KUKA KRL program: EPS_2_251315_MH01A_A_20251126070854.src

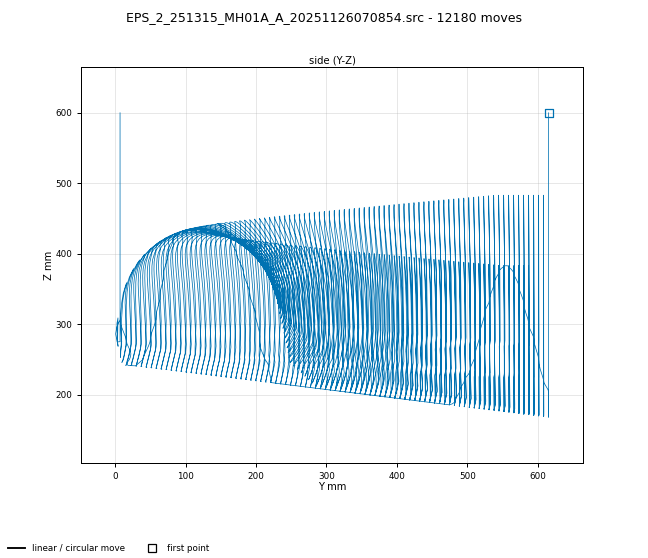
[picture p0: tool path of EPS_2_251315_MH01A_A_20251126070854.src, 12180 of 12182 moves have a stored position in this frame; points joined in program order, loops and branches not executed]
&ACCESS RVP
&REL 4
&COMMENT QRS 19112012
&PARAM EDITMASK = *
DEF PART()
EXT BAS (BAS_COMMAND :IN,REAL :IN )
INT I
BAS (#INITMOV,0 )

;KUKA QRS Post kuka4.cps  Date:22-06-2017 !

File_ID=2929

QRS_PRE_INIT()

;Init var - Until changes are made in qrs_pre_init
Outlet_Square_prg=0
Inlet_1_Square_prg=0
Inlet_2_Square_prg=0
Inlet_3_Square_prg=0
Inlet_4_Square_prg=0
Inlet_5_Square_prg=0

Outlet_1={X 0.000, Y 540.910, Z 382.500, B 0.000, E1 0.000 }
Inlet_1={X 0.000, Y 548.330, Z 308.000, B 0.000, E1 110.000 }
Outlet_1_type=201
Inlet_1_type=150
;QRS#1=Sidecore dimensions
;QRS#2=200-8" PVC SDR 35
;QRS#3=150-6" PVC SDR 28
;QRS#4=
;QRS#5=
;QRS#6=
;QRS#7=
;QRS#8=
;QRS#9=12-08 PSX
;QRS#10=10-06 PSX
;QRS#11=
;QRS#12=
;QRS#13=
;QRS#14=
;QRS#15=
;QRS#16=1220x127x762 2,5'
;QRS#17=EPS Height
;QRS#18=483
;QRS#19=*
;QRS#20= UPDATED VERSION 22-06-2017
;QRS#21=*
Outlet_Square=0100
Inlet_1_Square=070
Inlet_2_Square=0
Inlet_3_Square=0
Inlet_4_Square=0
Inlet_5_Square=0
Mill_Square=1
Outlet_Square_Prg=204
Inlet_1_Square_prg=203

QRS_INIT()

$ADVANCE=5

; T1
PTP {E1 173.696,E2 173.696}
PTP {X 0,Y 615.498,A -85,B 0,C 180,E1 173.696,E2 173.696,E3 0,E4 0,E5 0,E6 0}
QRS_SPEED_INIT()
LIN {X 0,Y 615.498,Z 600,A -85,B 0,C 180,E1 173.696,E2 173.696,E3 0,E4 0,E5 0,E6 0} C_VEL
LIN {X 0,Y 615.498,Z 213.72,A -85,B 0,C 180,E1 173.696,E2 173.696} C_VEL
LIN {X 0,Y 615.498,Z 205.494,A -85,B 0,C 180,E1 173.696,E2 173.696} C_VEL
LIN {X 0,Y 615.487,Z 203.734,A -85,B 0,C 180,E1 173.422,E2 173.422} C_VEL
LIN {X 0,Y 615.486,Z 220.973,A -85,B 0,C 180,E1 170.47,E2 170.47} C_VEL
LIN {X 0,Y 615.484,Z 223.487,A -85,B 0,C 180,E1 170.097,E2 170.097} C_VEL
LIN {X 0,Y 615.48,Z 225.832,A -85,B 0,C 180,E1 170.034,E2 170.034} C_VEL
LIN {X 0,Y 615.49,Z 299.844,A -85,B 0,C 180,E1 169.155,E2 169.155} C_VEL
LIN {X 0,Y 615.497,Z 309.209,A -85,B 0,C 180,E1 168.959,E2 168.959} C_VEL
LIN {X 0,Y 615.498,Z 318.215,A -85,B 0,C 180,E1 168.682,E2 168.682} C_VEL
LIN {X 0,Y 615.499,Z 327.343,A -85,B 0,C 180,E1 168.307,E2 168.307} C_VEL
LIN {X 0,Y 615.495,Z 338.158,A -85,B 0,C 180,E1 167.722,E2 167.722} C_VEL
LIN {X 0,Y 615.496,Z 346.444,A -85,B 0,C 180,E1 167.135,E2 167.135} C_VEL
LIN {X 0,Y 615.5,Z 354.141,A -85,B 0,C 180,E1 166.463,E2 166.463} C_VEL
LIN {X 0,Y 615.497,Z 360.745,A -85,B 0,C 180,E1 165.758,E2 165.758} C_VEL
LIN {X 0,Y 615.495,Z 366.931,A -85,B 0,C 180,E1 164.944,E2 164.944} C_VEL
LIN {X 0,Y 615.492,Z 372.054,A -85,B 0,C 180,E1 164.095,E2 164.095} C_VEL
LIN {X 0,Y 615.498,Z 376.623,A -85,B 0,C 180,E1 163.072,E2 163.072} C_VEL
LIN {X 0,Y 615.487,Z 379.784,A -85,B 0,C 180,E1 162.043,E2 162.043} C_VEL
LIN {X 0,Y 615.487,Z 381.203,A -85,B 0,C 180,E1 161.354,E2 161.354} C_VEL
LIN {X 0,Y 615.491,Z 382.08,A -85,B 0,C 180,E1 160.663,E2 160.663} C_VEL
LIN {X 0,Y 615.492,Z 382.389,A -85,B 0,C 180,E1 159.968,E2 159.968} C_VEL
LIN {X 0,Y 615.496,Z 382.089,A -85,B 0,C 180,E1 159.27,E2 159.27} C_VEL
LIN {X 0,Y 615.493,Z 381.22,A -85,B 0,C 180,E1 158.569,E2 158.569} C_VEL
LIN {X 0,Y 615.492,Z 379.266,A -85,B 0,C 180,E1 157.653,E2 157.653} C_VEL
LIN {X 0,Y 615.492,Z 376.497,A -85,B 0,C 180,E1 156.801,E2 156.801} C_VEL
LIN {X 0,Y 615.492,Z 371.558,A -85,B 0,C 180,E1 155.729,E2 155.729} C_VEL
LIN {X 0,Y 615.494,Z 366.205,A -85,B 0,C 180,E1 154.864,E2 154.864} C_VEL
LIN {X 0,Y 615.493,Z 360.324,A -85,B 0,C 180,E1 154.103,E2 154.103} C_VEL
LIN {X 0,Y 615.495,Z 353.723,A -85,B 0,C 180,E1 153.406,E2 153.406} C_VEL
LIN {X 0,Y 615.485,Z 344.747,A -85,B 0,C 180,E1 152.639,E2 152.639} C_VEL
LIN {X 0,Y 615.495,Z 335.257,A -85,B 0,C 180,E1 152.019,E2 152.019} C_VEL
LIN {X 0,Y 615.499,Z 326.105,A -85,B 0,C 180,E1 151.548,E2 151.548} C_VEL
LIN {X 0,Y 615.498,Z 317.502,A -85,B 0,C 180,E1 151.203,E2 151.203} C_VEL
LIN {X 0,Y 615.498,Z 308.063,A -85,B 0,C 180,E1 150.923,E2 150.923} C_VEL
LIN {X 0,Y 615.484,Z 298.594,A -85,B 0,C 180,E1 150.735,E2 150.735} C_VEL
LIN {X 0,Y 615.478,Z 223.968,A -85,B 0,C 180,E1 149.84,E2 149.84} C_VEL
LIN {X 0,Y 615.481,Z 222.831,A -85,B 0,C 180,E1 149.745,E2 149.745} C_VEL
LIN {X 0,Y 615.475,Z 206.472,A -85,B 0,C 180,E1 146.959,E2 146.959} C_VEL
LIN {X 0,Y 615.468,Z 191.559,A -85,B 0,C 180,E1 144.383,E2 144.383} C_VEL
LIN {X 0,Y 615.492,Z 175.153,A -85,B 0,C 180,E1 141.516,E2 141.516} C_VEL
LIN {X 0,Y 615.493,Z 167.764,A -85,B 0,C 180,E1 140.166,E2 140.166} C_VEL
LIN {X 0,Y 615.491,Z 167.686,A -85,B 0,C 180,E1 137.648,E2 137.648} C_VEL
LIN {X 0,Y 615.462,Z 167.69,A -85,B 0,C 180,E1 134.93,E2 134.93} C_VEL
LIN {X 0,Y 615.491,Z 167.695,A -85,B 0,C 180,E1 132.081,E2 132.081} C_VEL
LIN {X 0,Y 615.491,Z 167.686,A -85,B 0,C 180,E1 129.75,E2 129.75} C_VEL
LIN {X 0,Y 615.465,Z 167.691,A -85,B 0,C 180,E1 126.934,E2 126.934} C_VEL
LIN {X 0,Y 615.473,Z 167.695,A -85,B 0,C 180,E1 124.699,E2 124.699} C_VEL
LIN {X 0,Y 615.495,Z 167.698,A -85,B 0,C 180,E1 122.333,E2 122.333} C_VEL
LIN {X 0,Y 615.477,Z 167.685,A -85,B 0,C 180,E1 119.407,E2 119.407} C_VEL
LIN {X 0,Y 615.468,Z 167.691,A -85,B 0,C 180,E1 117.042,E2 117.042} C_VEL
LIN {X 0,Y 615.469,Z 167.693,A -85,B 0,C 180,E1 114.993,E2 114.993} C_VEL
LIN {X 0,Y 615.482,Z 167.69,A -85,B 0,C 180,E1 112.137,E2 112.137} C_VEL
LIN {X 0,Y 615.471,Z 167.688,A -85,B 0,C 180,E1 109.339,E2 109.339} C_VEL
LIN {X 0,Y 615.495,Z 167.698,A -85,B 0,C 180,E1 106.587,E2 106.587} C_VEL
LIN {X 0,Y 615.498,Z 167.681,A -85,B 0,C 180,E1 103.874,E2 103.874} C_VEL
LIN {X 0,Y 615.472,Z 167.692,A -85,B 0,C 180,E1 101.194,E2 101.194} C_VEL
LIN {X 0,Y 615.486,Z 167.694,A -85,B 0,C 180,E1 98.537,E2 98.537} C_VEL
LIN {X 0,Y 615.495,Z 167.681,A -85,B 0,C 180,E1 95.899,E2 95.899} C_VEL
LIN {X 0,Y 615.474,Z 167.693,A -85,B 0,C 180,E1 93.273,E2 93.273} C_VEL
LIN {X 0,Y 615.485,Z 167.694,A -85,B 0,C 180,E1 90.655,E2 90.655} C_VEL
LIN {X 0,Y 615.498,Z 167.68,A -85,B 0,C 180,E1 88.037,E2 88.037} C_VEL
LIN {X 0,Y 615.476,Z 167.692,A -85,B 0,C 180,E1 85.416,E2 85.416} C_VEL
LIN {X 0,Y 615.484,Z 167.695,A -85,B 0,C 180,E1 82.785,E2 82.785} C_VEL
LIN {X 0,Y 615.495,Z 167.681,A -85,B 0,C 180,E1 80.139,E2 80.139} C_VEL
LIN {X 0,Y 615.474,Z 167.694,A -85,B 0,C 180,E1 77.47,E2 77.47} C_VEL
LIN {X 0,Y 615.479,Z 167.692,A -85,B 0,C 180,E1 74.774,E2 74.774} C_VEL
LIN {X 0,Y 615.488,Z 167.683,A -85,B 0,C 180,E1 72.044,E2 72.044} C_VEL
LIN {X 0,Y 615.491,Z 167.701,A -85,B 0,C 180,E1 69.27,E2 69.27} C_VEL
LIN {X 0,Y 615.486,Z 167.683,A -85,B 0,C 180,E1 66.444,E2 66.444} C_VEL
LIN {X 0,Y 615.48,Z 167.696,A -85,B 0,C 180,E1 63.556,E2 63.556} C_VEL
LIN {X 0,Y 615.485,Z 167.703,A -85,B 0,C 180,E1 61.343,E2 61.343} C_VEL
LIN {X 0,Y 615.475,Z 167.691,A -85,B 0,C 180,E1 58.915,E2 58.915} C_VEL
LIN {X 0,Y 615.49,Z 167.682,A -85,B 0,C 180,E1 56.465,E2 56.465} C_VEL
LIN {X 0,Y 615.483,Z 167.7,A -85,B 0,C 180,E1 53.576,E2 53.576} C_VEL
LIN {X 0,Y 615.47,Z 167.69,A -85,B 0,C 180,E1 50.939,E2 50.939} C_VEL
LIN {X 0,Y 615.49,Z 167.682,A -85,B 0,C 180,E1 48.528,E2 48.528} C_VEL
LIN {X 0,Y 615.486,Z 167.695,A -85,B 0,C 180,E1 45.852,E2 45.852} C_VEL
LIN {X 0,Y 615.469,Z 167.69,A -85,B 0,C 180,E1 43.047,E2 43.047} C_VEL
LIN {X 0,Y 615.491,Z 167.682,A -85,B 0,C 180,E1 40.606,E2 40.606} C_VEL
LIN {X 0,Y 615.486,Z 167.693,A -85,B 0,C 180,E1 38.013,E2 38.013} C_VEL
LIN {X 0,Y 615.486,Z 167.698,A -85,B 0,C 180,E1 35.615,E2 35.615} C_VEL
LIN {X 0,Y 615.468,Z 167.691,A -85,B 0,C 180,E1 33.237,E2 33.237} C_VEL
LIN {X 0,Y 615.478,Z 167.685,A -85,B 0,C 180,E1 30.92,E2 30.92} C_VEL
LIN {X 0,Y 615.487,Z 167.686,A -85,B 0,C 180,E1 28.452,E2 28.452} C_VEL
LIN {X 0,Y 615.472,Z 167.694,A -85,B 0,C 180,E1 25.568,E2 25.568} C_VEL
LIN {X 0,Y 615.49,Z 167.682,A -85,B 0,C 180,E1 22.844,E2 22.844} C_VEL
LIN {X 0,Y 615.486,Z 167.702,A -85,B 0,C 180,E1 20.032,E2 20.032} C_VEL
LIN {X 0,Y 615.467,Z 167.688,A -85,B 0,C 180,E1 17.271,E2 17.271} C_VEL
LIN {X 0,Y 615.488,Z 167.688,A -85,B 0,C 180,E1 14.549,E2 14.549} C_VEL
LIN {X 0,Y 615.475,Z 167.696,A -85,B 0,C 180,E1 11.861,E2 11.861} C_VEL
LIN {X 0,Y 615.473,Z 167.686,A -85,B 0,C 180,E1 9.199,E2 9.199} C_VEL
LIN {X 0,Y 615.486,Z 167.692,A -85,B 0,C 180,E1 6.556,E2 6.556} C_VEL
LIN {X 0,Y 615.471,Z 167.695,A -85,B 0,C 180,E1 3.928,E2 3.928} C_VEL
LIN {X 0,Y 615.471,Z 167.686,A -85,B 0,C 180,E1 1.308,E2 1.308} C_VEL
LIN {X 0,Y 615.489,Z 167.691,A -85,B 0,C 180,E1 -1.309,E2 -1.309} C_VEL
LIN {X 0,Y 615.47,Z 167.696,A -85,B 0,C 180,E1 -3.929,E2 -3.929} C_VEL
LIN {X 0,Y 615.468,Z 167.687,A -85,B 0,C 180,E1 -6.571,E2 -6.571} C_VEL
LIN {X 0,Y 615.49,Z 167.691,A -85,B 0,C 180,E1 -9.199,E2 -9.199} C_VEL
LIN {X 0,Y 615.466,Z 167.695,A -85,B 0,C 180,E1 -11.862,E2 -11.862} C_VEL
LIN {X 0,Y 615.471,Z 167.686,A -85,B 0,C 180,E1 -14.55,E2 -14.55} C_VEL
LIN {X 0,Y 615.494,Z 167.696,A -85,B 0,C 180,E1 -17.271,E2 -17.271} C_VEL
LIN {X 0,Y 615.453,Z 167.693,A -85,B 0,C 180,E1 -20.034,E2 -20.034} C_VEL
LIN {X 0,Y 615.496,Z 167.686,A -85,B 0,C 180,E1 -22.845,E2 -22.845} C_VEL
LIN {X 0,Y 615.459,Z 167.695,A -85,B 0,C 180,E1 -25.717,E2 -25.717} C_VEL
LIN {X 0,Y 615.453,Z 167.692,A -85,B 0,C 180,E1 -27.917,E2 -27.917} C_VEL
LIN {X 0,Y 615.454,Z 167.69,A -85,B 0,C 180,E1 -30.162,E2 -30.162} C_VEL
LIN {X 0,Y 615.479,Z 167.686,A -85,B 0,C 180,E1 -32.458,E2 -32.458} C_VEL
LIN {X 0,Y 615.492,Z 167.691,A -85,B 0,C 180,E1 -34.815,E2 -34.815} C_VEL
LIN {X 0,Y 615.482,Z 167.699,A -85,B 0,C 180,E1 -37.243,E2 -37.243} C_VEL
LIN {X 0,Y 615.449,Z 167.693,A -85,B 0,C 180,E1 -39.753,E2 -39.753} C_VEL
LIN {X 0,Y 615.479,Z 167.687,A -85,B 0,C 180,E1 -42.354,E2 -42.354} C_VEL
LIN {X 0,Y 615.486,Z 167.699,A -85,B 0,C 180,E1 -45.069,E2 -45.069} C_VEL
LIN {X 0,Y 615.447,Z 167.693,A -85,B 0,C 180,E1 -47.645,E2 -47.645} C_VEL
LIN {X 0,Y 615.477,Z 167.688,A -85,B 0,C 180,E1 -50.25,E2 -50.25} C_VEL
LIN {X 0,Y 615.471,Z 167.699,A -85,B 0,C 180,E1 -53.066,E2 -53.066} C_VEL
LIN {X 0,Y 615.452,Z 167.696,A -85,B 0,C 180,E1 -55.305,E2 -55.305} C_VEL
LIN {X 0,Y 615.444,Z 167.692,A -85,B 0,C 180,E1 -57.676,E2 -57.676} C_VEL
LIN {X 0,Y 615.482,Z 167.688,A -85,B 0,C 180,E1 -60.207,E2 -60.207} C_VEL
LIN {X 0,Y 615.468,Z 167.698,A -85,B 0,C 180,E1 -62.959,E2 -62.959} C_VEL
LIN {X 0,Y 615.46,Z 167.697,A -85,B 0,C 180,E1 -65.008,E2 -65.008} C_VEL
LIN {X 0,Y 615.497,Z 167.805,A -85,B 0,C 180,E1 -66.712,E2 -66.712} C_VEL
LIN {X 0,Y 615.497,Z 168.158,A -85,B 0,C 180,E1 -66.801,E2 -66.801} C_VEL
LIN {X 0,Y 615.481,Z 193.361,A -85,B 0,C 180,E1 -69.445,E2 -69.445} C_VEL
LIN {X 0,Y 615.482,Z 220.3,A -85,B 0,C 180,E1 -72.215,E2 -72.215} C_VEL
LIN {X 0,Y 615.481,Z 247.213,A -85,B 0,C 180,E1 -74.944,E2 -74.944} C_VEL
LIN {X 0,Y 615.475,Z 268.865,A -85,B 0,C 180,E1 -77.093,E2 -77.093} C_VEL
LIN {X 0,Y 615.495,Z 378.861,A -85,B 0,C 180,E1 -78.411,E2 -78.411} C_VEL
LIN {X 0,Y 615.499,Z 391.363,A -85,B 0,C 180,E1 -78.683,E2 -78.683} C_VEL
LIN {X 0,Y 615.496,Z 404.501,A -85,B 0,C 180,E1 -79.109,E2 -79.109} C_VEL
LIN {X 0,Y 615.488,Z 416.488,A -85,B 0,C 180,E1 -79.64,E2 -79.64} C_VEL
LIN {X 0,Y 615.495,Z 428.002,A -85,B 0,C 180,E1 -80.304,E2 -80.304} C_VEL
LIN {X 0,Y 615.499,Z 438.348,A -85,B 0,C 180,E1 -81.05,E2 -81.05} C_VEL
LIN {X 0,Y 615.497,Z 446.817,A -85,B 0,C 180,E1 -81.795,E2 -81.795} C_VEL
LIN {X 0,Y 615.498,Z 454.611,A -85,B 0,C 180,E1 -82.62,E2 -82.62} C_VEL
LIN {X 0,Y 615.496,Z 462.206,A -85,B 0,C 180,E1 -83.609,E2 -83.609} C_VEL
LIN {X 0,Y 615.498,Z 469.207,A -85,B 0,C 180,E1 -84.759,E2 -84.759} C_VEL
LIN {X 0,Y 615.494,Z 473.853,A -85,B 0,C 180,E1 -85.744,E2 -85.744} C_VEL
LIN {X 0,Y 615.494,Z 477.4,A -85,B 0,C 180,E1 -86.728,E2 -86.728} C_VEL
LIN {X 0,Y 615.497,Z 479.234,A -85,B 0,C 180,E1 -87.383,E2 -87.383} C_VEL
LIN {X 0,Y 615.499,Z 480.608,A -85,B 0,C 180,E1 -88.037,E2 -88.037} C_VEL
LIN {X 0,Y 615.496,Z 482.174,A -85,B 0,C 180,E1 -89.346,E2 -89.346} C_VEL
LIN {X 0,Y 615.494,Z 482.389,A -85,B 0,C 180,E1 -90,E2 -90} C_VEL
LIN {X 0,Y 615.495,Z 481.579,A -85,B 0,C 180,E1 -91.309,E2 -91.309} C_VEL
LIN {X 0,Y 615.499,Z 480.607,A -85,B 0,C 180,E1 -91.963,E2 -91.963} C_VEL
LIN {X 0,Y 615.497,Z 479.232,A -85,B 0,C 180,E1 -92.618,E2 -92.618} C_VEL
LIN {X 0,Y 615.496,Z 476.348,A -85,B 0,C 180,E1 -93.601,E2 -93.601} C_VEL
LIN {X 0,Y 615.498,Z 472.44,A -85,B 0,C 180,E1 -94.585,E2 -94.585} C_VEL
LIN {X 0,Y 615.499,Z 467.403,A -85,B 0,C 180,E1 -95.57,E2 -95.57} C_VEL
LIN {X 0,Y 615.497,Z 460.87,A -85,B 0,C 180,E1 -96.583,E2 -96.583} C_VEL
LIN {X 0,Y 615.497,Z 453.13,A -85,B 0,C 180,E1 -97.546,E2 -97.546} C_VEL
LIN {X 0,Y 615.498,Z 445.041,A -85,B 0,C 180,E1 -98.372,E2 -98.372} C_VEL
LIN {X 0,Y 615.499,Z 435.162,A -85,B 0,C 180,E1 -99.199,E2 -99.199} C_VEL
LIN {X 0,Y 615.492,Z 423.974,A -85,B 0,C 180,E1 -99.945,E2 -99.945} C_VEL
LIN {X 0,Y 615.492,Z 413.014,A -85,B 0,C 180,E1 -100.527,E2 -100.527} C_VEL
LIN {X 0,Y 615.499,Z 400.411,A -85,B 0,C 180,E1 -101.042,E2 -101.042} C_VEL
LIN {X 0,Y 615.499,Z 388.047,A -85,B 0,C 180,E1 -101.402,E2 -101.402} C_VEL
LIN {X 0,Y 615.495,Z 374.439,A -85,B 0,C 180,E1 -101.652,E2 -101.652} C_VEL
LIN {X 0,Y 615.48,Z 268.847,A -85,B 0,C 180,E1 -102.908,E2 -102.908} C_VEL
LIN {X 0,Y 615.493,Z 243.842,A -85,B 0,C 180,E1 -105.396,E2 -105.396} C_VEL
LIN {X 0,Y 615.464,Z 215.482,A -85,B 0,C 180,E1 -108.277,E2 -108.277} C_VEL
LIN {X 0,Y 615.463,Z 189.975,A -85,B 0,C 180,E1 -110.907,E2 -110.907} C_VEL
LIN {X 0,Y 615.497,Z 168.024,A -85,B 0,C 180,E1 -113.222,E2 -113.222} C_VEL
LIN {X 0,Y 615.497,Z 167.694,A -85,B 0,C 180,E1 -113.556,E2 -113.556} C_VEL
LIN {X 0,Y 615.499,Z 167.687,A -85,B 0,C 180,E1 -115.715,E2 -115.715} C_VEL
LIN {X 0,Y 615.443,Z 167.693,A -85,B 0,C 180,E1 -118.442,E2 -118.442} C_VEL
LIN {X 0,Y 615.481,Z 167.699,A -85,B 0,C 180,E1 -121.084,E2 -121.084} C_VEL
LIN {X 0,Y 615.458,Z 167.69,A -85,B 0,C 180,E1 -124.024,E2 -124.024} C_VEL
LIN {X 0,Y 615.446,Z 167.694,A -85,B 0,C 180,E1 -126.428,E2 -126.428} C_VEL
LIN {X 0,Y 615.492,Z 167.7,A -85,B 0,C 180,E1 -129.062,E2 -129.062} C_VEL
LIN {X 0,Y 615.494,Z 167.688,A -85,B 0,C 180,E1 -131.473,E2 -131.473} C_VEL
LIN {X 0,Y 615.45,Z 167.691,A -85,B 0,C 180,E1 -134.153,E2 -134.153} C_VEL
LIN {X 0,Y 615.487,Z 167.703,A -85,B 0,C 180,E1 -136.953,E2 -136.953} C_VEL
LIN {X 0,Y 615.494,Z 167.687,A -85,B 0,C 180,E1 -139.394,E2 -139.394} C_VEL
LIN {X 0,Y 615.454,Z 167.69,A -85,B 0,C 180,E1 -141.992,E2 -141.992} C_VEL
LIN {X 0,Y 615.459,Z 167.695,A -85,B 0,C 180,E1 -144.382,E2 -144.382} C_VEL
LIN {X 0,Y 615.484,Z 167.703,A -85,B 0,C 180,E1 -146.763,E2 -146.763} C_VEL
LIN {X 0,Y 615.491,Z 167.691,A -85,B 0,C 180,E1 -149.08,E2 -149.08} C_VEL
LIN {X 0,Y 615.475,Z 167.686,A -85,B 0,C 180,E1 -151.552,E2 -151.552} C_VEL
LIN {X 0,Y 615.464,Z 167.696,A -85,B 0,C 180,E1 -154.283,E2 -154.283} C_VEL
LIN {X 0,Y 615.494,Z 167.685,A -85,B 0,C 180,E1 -157.155,E2 -157.155} C_VEL
LIN {X 0,Y 615.473,Z 167.686,A -85,B 0,C 180,E1 -159.446,E2 -159.446} C_VEL
LIN {X 0,Y 615.462,Z 167.693,A -85,B 0,C 180,E1 -162.042,E2 -162.042} C_VEL
LIN {X 0,Y 615.487,Z 167.693,A -85,B 0,C 180,E1 -164.774,E2 -164.774} C_VEL
LIN {X 0,Y 615.471,Z 167.686,A -85,B 0,C 180,E1 -167.469,E2 -167.469} C_VEL
LIN {X 0,Y 615.476,Z 167.696,A -85,B 0,C 180,E1 -170.137,E2 -170.137} C_VEL
LIN {X 0,Y 615.488,Z 167.689,A -85,B 0,C 180,E1 -172.784,E2 -172.784} C_VEL
LIN {X 0,Y 615.466,Z 167.688,A -85,B 0,C 180,E1 -175.415,E2 -175.415} C_VEL
LIN {X 0,Y 615.479,Z 167.697,A -85,B 0,C 180,E1 -178.037,E2 -178.037} C_VEL
LIN {X 0,Y 615.493,Z 167.889,A -85,B 0,C 180,E1 -180.306,E2 -180.306} C_VEL
LIN {X 0,Y 615.493,Z 182.783,A -85,B 0,C 180,E1 -182.945,E2 -182.945} C_VEL
LIN {X 0,Y 615.473,Z 199.791,A -85,B 0,C 180,E1 -185.898,E2 -185.898} C_VEL
LIN {X 0,Y 615.487,Z 203.734,A -85,B 0,C 180,E1 -186.578,E2 -186.578} C_VEL
LIN {X 0,Y 614.833,Z 206.671,A -85,B 0,C 180,E1 -187.055,E2 -187.055} C_VEL
LIN {X 0,Y 609.148,Z 216.391,A -85,B 0,C 180,E1 -188.585,E2 -188.585} C_VEL
LIN {X 0,Y 608.456,Z 219.26,A -85,B 0,C 180,E1 -189.067,E2 -189.067} C_VEL
LIN {X 0,Y 608.467,Z 223.705,A -85,B 0,C 180,E1 -189.788,E2 -189.788} C_VEL
LIN {X 0,Y 608.516,Z 226.354,A -85,B 0,C 180,E1 -189.85,E2 -189.85} C_VEL
LIN {X 0,Y 608.497,Z 299.098,A -85,B 0,C 180,E1 -190.718,E2 -190.718} C_VEL
LIN {X 0,Y 608.511,Z 308.516,A -85,B 0,C 180,E1 -190.91,E2 -190.91} C_VEL
LIN {X 0,Y 608.509,Z 317.848,A -85,B 0,C 180,E1 -191.192,E2 -191.192} C_VEL
LIN {X 0,Y 608.498,Z 325.357,A -85,B 0,C 180,E1 -191.492,E2 -191.492} C_VEL
LIN {X 0,Y 608.488,Z 333.777,A -85,B 0,C 180,E1 -191.914,E2 -191.914} C_VEL
LIN {X 0,Y 608.471,Z 341.913,A -85,B 0,C 180,E1 -192.422,E2 -192.422} C_VEL
LIN {X 0,Y 608.466,Z 349.663,A -85,B 0,C 180,E1 -193.016,E2 -193.016} C_VEL
LIN {X 0,Y 608.457,Z 356.947,A -85,B 0,C 180,E1 -193.697,E2 -193.697} C_VEL
LIN {X 0,Y 608.457,Z 364.237,A -85,B 0,C 180,E1 -194.55,E2 -194.55} C_VEL
LIN {X 0,Y 608.43,Z 369.982,A -85,B 0,C 180,E1 -195.407,E2 -195.407} C_VEL
LIN {X 0,Y 608.436,Z 373.737,A -85,B 0,C 180,E1 -196.094,E2 -196.094} C_VEL
LIN {X 0,Y 608.458,Z 376.808,A -85,B 0,C 180,E1 -196.784,E2 -196.784} C_VEL
LIN {X 0,Y 608.435,Z 379.203,A -85,B 0,C 180,E1 -197.477,E2 -197.477} C_VEL
LIN {X 0,Y 608.415,Z 380.952,A -85,B 0,C 180,E1 -198.173,E2 -198.173} C_VEL
LIN {X 0,Y 608.409,Z 382.146,A -85,B 0,C 180,E1 -198.871,E2 -198.871} C_VEL
LIN {X 0,Y 608.409,Z 382.802,A -85,B 0,C 180,E1 -199.572,E2 -199.572} C_VEL
LIN {X 0,Y 608.438,Z 382.73,A -85,B 0,C 180,E1 -200.671,E2 -200.671} C_VEL
LIN {X 0,Y 608.423,Z 381.457,A -85,B 0,C 180,E1 -201.693,E2 -201.693} C_VEL
LIN {X 0,Y 608.445,Z 378.686,A -85,B 0,C 180,E1 -202.764,E2 -202.764} C_VEL
LIN {X 0,Y 608.447,Z 376.076,A -85,B 0,C 180,E1 -203.484,E2 -203.484} C_VEL
LIN {X 0,Y 608.44,Z 372.061,A -85,B 0,C 180,E1 -204.323,E2 -204.323} C_VEL
LIN {X 0,Y 608.455,Z 367.232,A -85,B 0,C 180,E1 -205.118,E2 -205.118} C_VEL
LIN {X 0,Y 608.438,Z 361.973,A -85,B 0,C 180,E1 -205.823,E2 -205.823} C_VEL
LIN {X 0,Y 608.47,Z 354.964,A -85,B 0,C 180,E1 -206.588,E2 -206.588} C_VEL
LIN {X 0,Y 608.454,Z 348.097,A -85,B 0,C 180,E1 -207.203,E2 -207.203} C_VEL
LIN {X 0,Y 608.483,Z 340.037,A -85,B 0,C 180,E1 -207.796,E2 -207.796} C_VEL
LIN {X 0,Y 608.503,Z 330.616,A -85,B 0,C 180,E1 -208.353,E2 -208.353} C_VEL
LIN {X 0,Y 608.512,Z 319.962,A -85,B 0,C 180,E1 -208.824,E2 -208.824} C_VEL
LIN {X 0,Y 608.496,Z 310.259,A -85,B 0,C 180,E1 -209.136,E2 -209.136} C_VEL
LIN {X 0,Y 608.491,Z 300.482,A -85,B 0,C 180,E1 -209.35,E2 -209.35} C_VEL
LIN {X 0,Y 608.497,Z 239.342,A -85,B 0,C 180,E1 -210.088,E2 -210.088} C_VEL
LIN {X 0,Y 608.484,Z 224.05,A -85,B 0,C 180,E1 -210.281,E2 -210.281} C_VEL
LIN {X 0,Y 608.469,Z 223.023,A -85,B 0,C 180,E1 -210.383,E2 -210.383} C_VEL
LIN {X 0,Y 608.443,Z 206.2,A -85,B 0,C 180,E1 -213.275,E2 -213.275} C_VEL
LIN {X 0,Y 608.458,Z 191.372,A -85,B 0,C 180,E1 -215.856,E2 -215.856} C_VEL
LIN {X 0,Y 608.488,Z 175.892,A -85,B 0,C 180,E1 -218.586,E2 -218.586} C_VEL
LIN {X 0,Y 608.492,Z 168.769,A -85,B 0,C 180,E1 -219.894,E2 -219.894} C_VEL
LIN {X 0,Y 608.434,Z 168.69,A -85,B 0,C 180,E1 -222.961,E2 -222.961} C_VEL
LIN {X 0,Y 608.46,Z 168.697,A -85,B 0,C 180,E1 -225.735,E2 -225.735} C_VEL
LIN {X 0,Y 608.456,Z 168.687,A -85,B 0,C 180,E1 -228.658,E2 -228.658} C_VEL
LIN {X 0,Y 608.466,Z 168.695,A -85,B 0,C 180,E1 -231.759,E2 -231.759} C_VEL
LIN {X 0,Y 608.442,Z 168.689,A -85,B 0,C 180,E1 -234.722,E2 -234.722} C_VEL
LIN {X 0,Y 608.467,Z 168.694,A -85,B 0,C 180,E1 -237.476,E2 -237.476} C_VEL
LIN {X 0,Y 608.475,Z 168.686,A -85,B 0,C 180,E1 -240.221,E2 -240.221} C_VEL
LIN {X 0,Y 608.464,Z 168.687,A -85,B 0,C 180,E1 -242.795,E2 -242.795} C_VEL
LIN {X 0,Y 608.447,Z 168.698,A -85,B 0,C 180,E1 -245.428,E2 -245.428} C_VEL
LIN {X 0,Y 608.46,Z 168.686,A -85,B 0,C 180,E1 -248.308,E2 -248.308} C_VEL
LIN {X 0,Y 608.453,Z 168.694,A -85,B 0,C 180,E1 -251.13,E2 -251.13} C_VEL
LIN {X 0,Y 608.462,Z 168.688,A -85,B 0,C 180,E1 -253.906,E2 -253.906} C_VEL
LIN {X 0,Y 608.456,Z 168.688,A -85,B 0,C 180,E1 -256.643,E2 -256.643} C_VEL
LIN {X 0,Y 608.465,Z 168.695,A -85,B 0,C 180,E1 -259.35,E2 -259.35} C_VEL
LIN {X 0,Y 608.478,Z 168.684,A -85,B 0,C 180,E1 -262.033,E2 -262.033} C_VEL
LIN {X 0,Y 608.456,Z 168.69,A -85,B 0,C 180,E1 -264.698,E2 -264.698} C_VEL
LIN {X 0,Y 608.474,Z 168.691,A -85,B 0,C 180,E1 -267.352,E2 -267.352} C_VEL
LIN {X 0,Y 608.477,Z 168.684,A -85,B 0,C 180,E1 -270,E2 -270} C_VEL
LIN {X 0,Y 608.467,Z 168.69,A -85,B 0,C 180,E1 -272.648,E2 -272.648} C_VEL
LIN {X 0,Y 608.462,Z 168.691,A -85,B 0,C 180,E1 -275.301,E2 -275.301} C_VEL
LIN {X 0,Y 608.477,Z 168.684,A -85,B 0,C 180,E1 -277.966,E2 -277.966} C_VEL
LIN {X 0,Y 608.459,Z 168.693,A -85,B 0,C 180,E1 -280.649,E2 -280.649} C_VEL
LIN {X 0,Y 608.462,Z 168.689,A -85,B 0,C 180,E1 -283.356,E2 -283.356} C_VEL
LIN {X 0,Y 608.457,Z 168.687,A -85,B 0,C 180,E1 -286.093,E2 -286.093} C_VEL
LIN {X 0,Y 608.451,Z 168.697,A -85,B 0,C 180,E1 -288.869,E2 -288.869} C_VEL
LIN {X 0,Y 608.461,Z 168.686,A -85,B 0,C 180,E1 -291.691,E2 -291.691} C_VEL
LIN {X 0,Y 608.445,Z 168.697,A -85,B 0,C 180,E1 -294.571,E2 -294.571} C_VEL
LIN {X 0,Y 608.47,Z 168.687,A -85,B 0,C 180,E1 -297.207,E2 -297.207} C_VEL
LIN {X 0,Y 608.467,Z 168.687,A -85,B 0,C 180,E1 -299.972,E2 -299.972} C_VEL
LIN {X 0,Y 608.46,Z 168.696,A -85,B 0,C 180,E1 -302.523,E2 -302.523} C_VEL
LIN {X 0,Y 608.446,Z 168.689,A -85,B 0,C 180,E1 -305.276,E2 -305.276} C_VEL
LIN {X 0,Y 608.463,Z 168.687,A -85,B 0,C 180,E1 -307.746,E2 -307.746} C_VEL
LIN {X 0,Y 608.449,Z 168.696,A -85,B 0,C 180,E1 -310.329,E2 -310.329} C_VEL
LIN {X 0,Y 608.442,Z 168.691,A -85,B 0,C 180,E1 -312.96,E2 -312.96} C_VEL
LIN {X 0,Y 608.448,Z 168.689,A -85,B 0,C 180,E1 -315.736,E2 -315.736} C_VEL
LIN {X 0,Y 608.452,Z 168.692,A -85,B 0,C 180,E1 -318.657,E2 -318.657} C_VEL
LIN {X 0,Y 608.46,Z 168.687,A -85,B 0,C 180,E1 -321.412,E2 -321.412} C_VEL
LIN {X 0,Y 608.472,Z 168.691,A -85,B 0,C 180,E1 -323.95,E2 -323.95} C_VEL
LIN {X 0,Y 608.458,Z 168.695,A -85,B 0,C 180,E1 -326.329,E2 -326.329} C_VEL
LIN {X 0,Y 608.467,Z 168.688,A -85,B 0,C 180,E1 -328.727,E2 -328.727} C_VEL
LIN {X 0,Y 608.473,Z 168.685,A -85,B 0,C 180,E1 -331.378,E2 -331.378} C_VEL
LIN {X 0,Y 608.463,Z 168.693,A -85,B 0,C 180,E1 -334.279,E2 -334.279} C_VEL
LIN {X 0,Y 608.446,Z 168.688,A -85,B 0,C 180,E1 -336.876,E2 -336.876} C_VEL
LIN {X 0,Y 608.462,Z 168.692,A -85,B 0,C 180,E1 -339.726,E2 -339.726} C_VEL
LIN {X 0,Y 608.44,Z 168.691,A -85,B 0,C 180,E1 -342.523,E2 -342.523} C_VEL
LIN {X 0,Y 608.471,Z 168.687,A -85,B 0,C 180,E1 -345.28,E2 -345.28} C_VEL
LIN {X 0,Y 608.453,Z 168.696,A -85,B 0,C 180,E1 -348,E2 -348} C_VEL
LIN {X 0,Y 608.457,Z 168.687,A -85,B 0,C 180,E1 -350.694,E2 -350.694} C_VEL
LIN {X 0,Y 608.468,Z 168.689,A -85,B 0,C 180,E1 -353.368,E2 -353.368} C_VEL
LIN {X 0,Y 608.441,Z 168.694,A -85,B 0,C 180,E1 -356.026,E2 -356.026} C_VEL
LIN {X 0,Y 608.455,Z 168.687,A -85,B 0,C 180,E1 -358.677,E2 -358.677} C_VEL
LIN {X 0,Y 608.472,Z 168.69,A -85,B 0,C 180,E1 -361.324,E2 -361.324} C_VEL
LIN {X 0,Y 608.438,Z 168.694,A -85,B 0,C 180,E1 -363.974,E2 -363.974} C_VEL
LIN {X 0,Y 608.451,Z 168.688,A -85,B 0,C 180,E1 -366.633,E2 -366.633} C_VEL
LIN {X 0,Y 608.47,Z 168.692,A -85,B 0,C 180,E1 -369.306,E2 -369.306} C_VEL
LIN {X 0,Y 608.444,Z 168.691,A -85,B 0,C 180,E1 -372,E2 -372} C_VEL
LIN {X 0,Y 608.465,Z 168.687,A -85,B 0,C 180,E1 -374.721,E2 -374.721} C_VEL
LIN {X 0,Y 608.449,Z 168.697,A -85,B 0,C 180,E1 -377.477,E2 -377.477} C_VEL
LIN {X 0,Y 608.44,Z 168.689,A -85,B 0,C 180,E1 -380.275,E2 -380.275} C_VEL
LIN {X 0,Y 608.451,Z 168.688,A -85,B 0,C 180,E1 -382.477,E2 -382.477} C_VEL
LIN {X 0,Y 608.445,Z 168.699,A -85,B 0,C 180,E1 -385.302,E2 -385.302} C_VEL
LIN {X 0,Y 608.436,Z 168.695,A -85,B 0,C 180,E1 -387.519,E2 -387.519} C_VEL
LIN {X 0,Y 608.437,Z 168.69,A -85,B 0,C 180,E1 -389.968,E2 -389.968} C_VEL
LIN {X 0,Y 608.454,Z 168.688,A -85,B 0,C 180,E1 -392.523,E2 -392.523} C_VEL
LIN {X 0,Y 608.428,Z 168.698,A -85,B 0,C 180,E1 -395.279,E2 -395.279} C_VEL
LIN {X 0,Y 608.447,Z 168.689,A -85,B 0,C 180,E1 -397.748,E2 -397.748} C_VEL
LIN {X 0,Y 608.439,Z 168.69,A -85,B 0,C 180,E1 -400.329,E2 -400.329} C_VEL
LIN {X 0,Y 608.46,Z 168.692,A -85,B 0,C 180,E1 -403.309,E2 -403.309} C_VEL
LIN {X 0,Y 608.446,Z 168.688,A -85,B 0,C 180,E1 -406.13,E2 -406.13} C_VEL
LIN {X 0,Y 608.458,Z 168.696,A -85,B 0,C 180,E1 -408.825,E2 -408.825} C_VEL
LIN {X 0,Y 608.422,Z 168.694,A -85,B 0,C 180,E1 -411.41,E2 -411.41} C_VEL
LIN {X 0,Y 608.437,Z 168.689,A -85,B 0,C 180,E1 -413.956,E2 -413.956} C_VEL
LIN {X 0,Y 608.461,Z 168.69,A -85,B 0,C 180,E1 -416.33,E2 -416.33} C_VEL
LIN {X 0,Y 608.444,Z 168.699,A -85,B 0,C 180,E1 -418.733,E2 -418.733} C_VEL
LIN {X 0,Y 608.437,Z 168.691,A -85,B 0,C 180,E1 -421.387,E2 -421.387} C_VEL
LIN {X 0,Y 608.433,Z 168.691,A -85,B 0,C 180,E1 -423.965,E2 -423.965} C_VEL
LIN {X 0,Y 608.522,Z 168.883,A -85,B 0,C 180,E1 -426.587,E2 -426.587} C_VEL
LIN {X 0,Y 608.66,Z 175.938,A -85,B 0,C 180,E1 -427.363,E2 -427.363} C_VEL
LIN {X 0,Y 608.599,Z 203.46,A -85,B 0,C 180,E1 -430.259,E2 -430.259} C_VEL
LIN {X 0,Y 608.547,Z 232.097,A -85,B 0,C 180,E1 -433.219,E2 -433.219} C_VEL
LIN {X 0,Y 608.504,Z 260.426,A -85,B 0,C 180,E1 -436.103,E2 -436.103} C_VEL
LIN {X 0,Y 608.515,Z 268.904,A -85,B 0,C 180,E1 -436.943,E2 -436.943} C_VEL
LIN {X 0,Y 608.546,Z 378.979,A -85,B 0,C 180,E1 -438.277,E2 -438.277} C_VEL
LIN {X 0,Y 608.547,Z 392.238,A -85,B 0,C 180,E1 -438.573,E2 -438.573} C_VEL
LIN {X 0,Y 608.544,Z 405.338,A -85,B 0,C 180,E1 -439.009,E2 -439.009} C_VEL
LIN {X 0,Y 608.509,Z 416.646,A -85,B 0,C 180,E1 -439.52,E2 -439.52} C_VEL
LIN {X 0,Y 608.486,Z 428.206,A -85,B 0,C 180,E1 -440.192,E2 -440.192} C_VEL
LIN {X 0,Y 608.485,Z 438.601,A -85,B 0,C 180,E1 -440.946,E2 -440.946} C_VEL
LIN {X 0,Y 608.475,Z 447.118,A -85,B 0,C 180,E1 -441.699,E2 -441.699} C_VEL
LIN {X 0,Y 608.47,Z 454.965,A -85,B 0,C 180,E1 -442.534,E2 -442.534} C_VEL
LIN {X 0,Y 608.46,Z 462.289,A -85,B 0,C 180,E1 -443.485,E2 -443.485} C_VEL
LIN {X 0,Y 608.45,Z 467.869,A -85,B 0,C 180,E1 -444.366,E2 -444.366} C_VEL
LIN {X 0,Y 608.432,Z 472.952,A -85,B 0,C 180,E1 -445.363,E2 -445.363} C_VEL
LIN {X 0,Y 608.449,Z 476.898,A -85,B 0,C 180,E1 -446.358,E2 -446.358} C_VEL
LIN {X 0,Y 608.425,Z 479.81,A -85,B 0,C 180,E1 -447.352,E2 -447.352} C_VEL
LIN {X 0,Y 608.444,Z 481.202,A -85,B 0,C 180,E1 -448.015,E2 -448.015} C_VEL
LIN {X 0,Y 608.438,Z 482.784,A -85,B 0,C 180,E1 -449.339,E2 -449.339} C_VEL
LIN {X 0,Y 608.434,Z 483,A -85,B 0,C 180,E1 -450,E2 -450} C_VEL
LIN {X 0,Y 608.448,Z 482.183,A -85,B 0,C 180,E1 -451.324,E2 -451.324} C_VEL
LIN {X 0,Y 608.444,Z 481.201,A -85,B 0,C 180,E1 -451.986,E2 -451.986} C_VEL
LIN {X 0,Y 608.425,Z 479.808,A -85,B 0,C 180,E1 -452.649,E2 -452.649} C_VEL
LIN {X 0,Y 608.449,Z 476.895,A -85,B 0,C 180,E1 -453.643,E2 -453.643} C_VEL
LIN {X 0,Y 608.432,Z 472.948,A -85,B 0,C 180,E1 -454.638,E2 -454.638} C_VEL
LIN {X 0,Y 608.437,Z 466.874,A -85,B 0,C 180,E1 -455.801,E2 -455.801} C_VEL
LIN {X 0,Y 608.462,Z 460.232,A -85,B 0,C 180,E1 -456.8,E2 -456.8} C_VEL
LIN {X 0,Y 608.456,Z 451.986,A -85,B 0,C 180,E1 -457.801,E2 -457.801} C_VEL
LIN {X 0,Y 608.472,Z 443.532,A -85,B 0,C 180,E1 -458.636,E2 -458.636} C_VEL
LIN {X 0,Y 608.479,Z 433.086,A -85,B 0,C 180,E1 -459.474,E2 -459.474} C_VEL
LIN {X 0,Y 608.496,Z 422.75,A -85,B 0,C 180,E1 -460.145,E2 -460.145} C_VEL
LIN {X 0,Y 608.523,Z 411.234,A -85,B 0,C 180,E1 -460.741,E2 -460.741} C_VEL
LIN {X 0,Y 608.541,Z 398.866,A -85,B 0,C 180,E1 -461.225,E2 -461.225} C_VEL
LIN {X 0,Y 608.549,Z 385.423,A -85,B 0,C 180,E1 -461.597,E2 -461.597} C_VEL
LIN {X 0,Y 608.552,Z 373.057,A -85,B 0,C 180,E1 -461.808,E2 -461.808} C_VEL
LIN {X 0,Y 608.517,Z 268.887,A -85,B 0,C 180,E1 -463.058,E2 -463.058} C_VEL
LIN {X 0,Y 608.539,Z 242.194,A -85,B 0,C 180,E1 -465.748,E2 -465.748} C_VEL
LIN {X 0,Y 608.554,Z 214.352,A -85,B 0,C 180,E1 -468.61,E2 -468.61} C_VEL
LIN {X 0,Y 608.587,Z 189.975,A -85,B 0,C 180,E1 -471.154,E2 -471.154} C_VEL
LIN {X 0,Y 608.671,Z 169.761,A -85,B 0,C 180,E1 -473.295,E2 -473.295} C_VEL
LIN {X 0,Y 608.499,Z 168.792,A -85,B 0,C 180,E1 -473.437,E2 -473.437} C_VEL
LIN {X 0,Y 608.433,Z 168.691,A -85,B 0,C 180,E1 -476.036,E2 -476.036} C_VEL
LIN {X 0,Y 608.438,Z 168.691,A -85,B 0,C 180,E1 -478.613,E2 -478.613} C_VEL
LIN {X 0,Y 608.448,Z 168.697,A -85,B 0,C 180,E1 -481.318,E2 -481.318} C_VEL
LIN {X 0,Y 608.449,Z 168.69,A -85,B 0,C 180,E1 -483.731,E2 -483.731} C_VEL
LIN {X 0,Y 608.438,Z 168.689,A -85,B 0,C 180,E1 -486.093,E2 -486.093} C_VEL
LIN {X 0,Y 608.422,Z 168.694,A -85,B 0,C 180,E1 -488.592,E2 -488.592} C_VEL
LIN {X 0,Y 608.467,Z 168.691,A -85,B 0,C 180,E1 -491.342,E2 -491.342} C_VEL
LIN {X 0,Y 608.448,Z 168.688,A -85,B 0,C 180,E1 -493.871,E2 -493.871} C_VEL
LIN {X 0,Y 608.464,Z 168.692,A -85,B 0,C 180,E1 -496.692,E2 -496.692} C_VEL
LIN {X 0,Y 608.455,Z 168.688,A -85,B 0,C 180,E1 -499.697,E2 -499.697} C_VEL
LIN {X 0,Y 608.481,Z 168.695,A -85,B 0,C 180,E1 -502.84,E2 -502.84} C_VEL
LIN {X 0,Y 608.465,Z 168.687,A -85,B 0,C 180,E1 -505.53,E2 -505.53} C_VEL
LIN {X 0,Y 608.449,Z 168.688,A -85,B 0,C 180,E1 -507.904,E2 -507.904} C_VEL
LIN {X 0,Y 608.443,Z 168.691,A -85,B 0,C 180,E1 -510.219,E2 -510.219} C_VEL
LIN {X 0,Y 608.482,Z 168.693,A -85,B 0,C 180,E1 -512.792,E2 -512.792} C_VEL
LIN {X 0,Y 608.443,Z 168.689,A -85,B 0,C 180,E1 -515.428,E2 -515.428} C_VEL
LIN {X 0,Y 608.464,Z 168.692,A -85,B 0,C 180,E1 -518.308,E2 -518.308} C_VEL
LIN {X 0,Y 608.467,Z 168.686,A -85,B 0,C 180,E1 -521.285,E2 -521.285} C_VEL
LIN {X 0,Y 608.443,Z 168.69,A -85,B 0,C 180,E1 -523.905,E2 -523.905} C_VEL
LIN {X 0,Y 608.462,Z 168.694,A -85,B 0,C 180,E1 -526.643,E2 -526.643} C_VEL
LIN {X 0,Y 608.455,Z 168.687,A -85,B 0,C 180,E1 -529.35,E2 -529.35} C_VEL
LIN {X 0,Y 608.469,Z 168.69,A -85,B 0,C 180,E1 -532.033,E2 -532.033} C_VEL
LIN {X 0,Y 608.467,Z 168.69,A -85,B 0,C 180,E1 -534.698,E2 -534.698} C_VEL
LIN {X 0,Y 608.465,Z 168.686,A -85,B 0,C 180,E1 -537.352,E2 -537.352} C_VEL
LIN {X 0,Y 608.47,Z 168.778,A -85,B 0,C 180,E1 -540.206,E2 -540.206} C_VEL
LIN {X 0,Y 608.487,Z 182.348,A -85,B 0,C 180,E1 -542.648,E2 -542.648} C_VEL
LIN {X 0,Y 608.439,Z 199.396,A -85,B 0,C 180,E1 -545.634,E2 -545.634} C_VEL
LIN {X 0,Y 608.44,Z 214.81,A -85,B 0,C 180,E1 -548.301,E2 -548.301} C_VEL
LIN {X 0,Y 608.456,Z 219.26,A -85,B 0,C 180,E1 -549.067,E2 -549.067} C_VEL
LIN {X 0,Y 608.101,Z 221.608,A -85,B 0,C 180,E1 -549.346,E2 -549.346} C_VEL
LIN {X 0,Y 607.284,Z 224.629,A -85,B 0,C 180,E1 -549.555,E2 -549.555} C_VEL
LIN {X 0,Y 605.599,Z 229.867,A -85,B 0,C 180,E1 -549.761,E2 -549.761} C_VEL
LIN {X 0,Y 603.731,Z 235.7,A -85,B 0,C 180,E1 -549.867,E2 -549.867} C_VEL
LIN {X 0,Y 601.822,Z 243.927,A -85,B 0,C 180,E1 -549.944,E2 -549.944} C_VEL
LIN {X 0,Y 601.523,Z 248.122,A -85,B 0,C 180,E1 -549.989,E2 -549.989} C_VEL
LIN {X 0,Y 601.508,Z 300.112,A -85,B 0,C 180,E1 -550.625,E2 -550.625} C_VEL
LIN {X 0,Y 601.496,Z 309.673,A -85,B 0,C 180,E1 -550.832,E2 -550.832} C_VEL
LIN {X 0,Y 601.506,Z 320.45,A -85,B 0,C 180,E1 -551.18,E2 -551.18} C_VEL
LIN {X 0,Y 601.449,Z 331.94,A -85,B 0,C 180,E1 -551.714,E2 -551.714} C_VEL
LIN {X 0,Y 601.414,Z 340.408,A -85,B 0,C 180,E1 -552.228,E2 -552.228} C_VEL
LIN {X 0,Y 601.406,Z 348.402,A -85,B 0,C 180,E1 -552.828,E2 -552.828} C_VEL
LIN {X 0,Y 601.382,Z 355.885,A -85,B 0,C 180,E1 -553.516,E2 -553.516} C_VEL
LIN {X 0,Y 601.382,Z 363.463,A -85,B 0,C 180,E1 -554.379,E2 -554.379} C_VEL
LIN {X 0,Y 601.356,Z 369.374,A -85,B 0,C 180,E1 -555.245,E2 -555.245} C_VEL
LIN {X 0,Y 601.354,Z 373.251,A -85,B 0,C 180,E1 -555.94,E2 -555.94} C_VEL
LIN {X 0,Y 601.357,Z 377.642,A -85,B 0,C 180,E1 -556.988,E2 -556.988} C_VEL
LIN {X 0,Y 601.321,Z 379.855,A -85,B 0,C 180,E1 -557.69,E2 -557.69} C_VEL
LIN {X 0,Y 601.316,Z 381.486,A -85,B 0,C 180,E1 -558.395,E2 -558.395} C_VEL
LIN {X 0,Y 601.301,Z 382.491,A -85,B 0,C 180,E1 -559.102,E2 -559.102} C_VEL
LIN {X 0,Y 601.308,Z 382.916,A -85,B 0,C 180,E1 -559.812,E2 -559.812} C_VEL
LIN {X 0,Y 601.338,Z 382.685,A -85,B 0,C 180,E1 -560.775,E2 -560.775} C_VEL
LIN {X 0,Y 601.34,Z 380.901,A -85,B 0,C 180,E1 -561.962,E2 -561.962} C_VEL
LIN {X 0,Y 601.34,Z 379.066,A -85,B 0,C 180,E1 -562.685,E2 -562.685} C_VEL
LIN {X 0,Y 601.345,Z 376.551,A -85,B 0,C 180,E1 -563.413,E2 -563.413} C_VEL
LIN {X 0,Y 601.369,Z 372.597,A -85,B 0,C 180,E1 -564.278,E2 -564.278} C_VEL
LIN {X 0,Y 601.375,Z 366.731,A -85,B 0,C 180,E1 -565.249,E2 -565.249} C_VEL
LIN {X 0,Y 601.394,Z 360.622,A -85,B 0,C 180,E1 -566.051,E2 -566.051} C_VEL
LIN {X 0,Y 601.395,Z 354.229,A -85,B 0,C 180,E1 -566.738,E2 -566.738} C_VEL
LIN {X 0,Y 601.409,Z 346.434,A -85,B 0,C 180,E1 -567.425,E2 -567.425} C_VEL
LIN {X 0,Y 601.459,Z 335.926,A -85,B 0,C 180,E1 -568.149,E2 -568.149} C_VEL
LIN {X 0,Y 601.478,Z 327.001,A -85,B 0,C 180,E1 -568.624,E2 -568.624} C_VEL
LIN {X 0,Y 601.485,Z 318.424,A -85,B 0,C 180,E1 -568.982,E2 -568.982} C_VEL
LIN {X 0,Y 601.516,Z 309.076,A -85,B 0,C 180,E1 -569.273,E2 -569.273} C_VEL
LIN {X 0,Y 601.505,Z 300.409,A -85,B 0,C 180,E1 -569.46,E2 -569.46} C_VEL
LIN {X 0,Y 601.449,Z 224.307,A -85,B 0,C 180,E1 -570.392,E2 -570.392} C_VEL
LIN {X 0,Y 601.398,Z 223.034,A -85,B 0,C 180,E1 -570.504,E2 -570.504} C_VEL
LIN {X 0,Y 601.404,Z 206.874,A -85,B 0,C 180,E1 -573.315,E2 -573.315} C_VEL
LIN {X 0,Y 601.439,Z 191.579,A -85,B 0,C 180,E1 -576.009,E2 -576.009} C_VEL
LIN {X 0,Y 601.511,Z 176.142,A -85,B 0,C 180,E1 -578.764,E2 -578.764} C_VEL
LIN {X 0,Y 601.463,Z 169.68,A -85,B 0,C 180,E1 -579.959,E2 -579.959} C_VEL
LIN {X 0,Y 601.406,Z 169.566,A -85,B 0,C 180,E1 -582.67,E2 -582.67} C_VEL
LIN {X 0,Y 601.425,Z 169.569,A -85,B 0,C 180,E1 -585.482,E2 -585.482} C_VEL
LIN {X 0,Y 601.422,Z 169.564,A -85,B 0,C 180,E1 -588.406,E2 -588.406} C_VEL
LIN {X 0,Y 601.427,Z 169.57,A -85,B 0,C 180,E1 -591.529,E2 -591.529} C_VEL
LIN {X 0,Y 601.406,Z 169.567,A -85,B 0,C 180,E1 -594.246,E2 -594.246} C_VEL
LIN {X 0,Y 601.425,Z 169.563,A -85,B 0,C 180,E1 -596.686,E2 -596.686} C_VEL
LIN {X 0,Y 601.408,Z 169.568,A -85,B 0,C 180,E1 -599.057,E2 -599.057} C_VEL
LIN {X 0,Y 601.431,Z 169.57,A -85,B 0,C 180,E1 -601.373,E2 -601.373} C_VEL
LIN {X 0,Y 601.419,Z 169.565,A -85,B 0,C 180,E1 -604.131,E2 -604.131} C_VEL
LIN {X 0,Y 601.417,Z 169.564,A -85,B 0,C 180,E1 -606.589,E2 -606.589} C_VEL
LIN {X 0,Y 601.431,Z 169.571,A -85,B 0,C 180,E1 -609.478,E2 -609.478} C_VEL
LIN {X 0,Y 601.393,Z 169.567,A -85,B 0,C 180,E1 -612.311,E2 -612.311} C_VEL
LIN {X 0,Y 601.407,Z 169.565,A -85,B 0,C 180,E1 -614.408,E2 -614.408} C_VEL
LIN {X 0,Y 601.418,Z 169.572,A -85,B 0,C 180,E1 -617.171,E2 -617.171} C_VEL
LIN {X 0,Y 601.439,Z 169.562,A -85,B 0,C 180,E1 -619.905,E2 -619.905} C_VEL
LIN {X 0,Y 601.435,Z 169.563,A -85,B 0,C 180,E1 -622.614,E2 -622.614} C_VEL
LIN {X 0,Y 601.421,Z 169.571,A -85,B 0,C 180,E1 -625.308,E2 -625.308} C_VEL
LIN {X 0,Y 601.437,Z 169.561,A -85,B 0,C 180,E1 -627.991,E2 -627.991} C_VEL
LIN {X 0,Y 601.442,Z 169.565,A -85,B 0,C 180,E1 -630.669,E2 -630.669} C_VEL
LIN {X 0,Y 601.429,Z 169.567,A -85,B 0,C 180,E1 -633.349,E2 -633.349} C_VEL
LIN {X 0,Y 601.437,Z 169.561,A -85,B 0,C 180,E1 -636.036,E2 -636.036} C_VEL
LIN {X 0,Y 601.409,Z 169.572,A -85,B 0,C 180,E1 -638.737,E2 -638.737} C_VEL
LIN {X 0,Y 601.432,Z 169.564,A -85,B 0,C 180,E1 -641.458,E2 -641.458} C_VEL
LIN {X 0,Y 601.416,Z 169.565,A -85,B 0,C 180,E1 -644.205,E2 -644.205} C_VEL
LIN {X 0,Y 601.428,Z 169.57,A -85,B 0,C 180,E1 -646.985,E2 -646.985} C_VEL
LIN {X 0,Y 601.4,Z 169.566,A -85,B 0,C 180,E1 -649.809,E2 -649.809} C_VEL
LIN {X 0,Y 601.411,Z 169.573,A -85,B 0,C 180,E1 -652.605,E2 -652.605} C_VEL
LIN {X 0,Y 601.397,Z 169.574,A -85,B 0,C 180,E1 -654.878,E2 -654.878} C_VEL
LIN {X 0,Y 601.417,Z 169.564,A -85,B 0,C 180,E1 -657.867,E2 -657.867} C_VEL
LIN {X 0,Y 601.423,Z 169.566,A -85,B 0,C 180,E1 -660.163,E2 -660.163} C_VEL
LIN {X 0,Y 601.419,Z 169.572,A -85,B 0,C 180,E1 -662.716,E2 -662.716} C_VEL
LIN {X 0,Y 601.41,Z 169.567,A -85,B 0,C 180,E1 -665.115,E2 -665.115} C_VEL
LIN {X 0,Y 601.428,Z 169.562,A -85,B 0,C 180,E1 -667.419,E2 -667.419} C_VEL
LIN {X 0,Y 601.406,Z 169.568,A -85,B 0,C 180,E1 -669.994,E2 -669.994} C_VEL
LIN {X 0,Y 601.407,Z 169.571,A -85,B 0,C 180,E1 -672.67,E2 -672.67} C_VEL
LIN {X 0,Y 601.418,Z 169.564,A -85,B 0,C 180,E1 -675.482,E2 -675.482} C_VEL
LIN {X 0,Y 601.417,Z 169.573,A -85,B 0,C 180,E1 -678.406,E2 -678.406} C_VEL
LIN {X 0,Y 601.426,Z 169.565,A -85,B 0,C 180,E1 -680.875,E2 -680.875} C_VEL
LIN {X 0,Y 601.437,Z 169.564,A -85,B 0,C 180,E1 -683.733,E2 -683.733} C_VEL
LIN {X 0,Y 601.419,Z 169.566,A -85,B 0,C 180,E1 -686.686,E2 -686.686} C_VEL
LIN {X 0,Y 601.422,Z 169.563,A -85,B 0,C 180,E1 -689.059,E2 -689.059} C_VEL
LIN {X 0,Y 601.432,Z 169.563,A -85,B 0,C 180,E1 -691.374,E2 -691.374} C_VEL
LIN {X 0,Y 601.407,Z 169.575,A -85,B 0,C 180,E1 -694.132,E2 -694.132} C_VEL
LIN {X 0,Y 601.416,Z 169.566,A -85,B 0,C 180,E1 -696.59,E2 -696.59} C_VEL
LIN {X 0,Y 601.43,Z 169.565,A -85,B 0,C 180,E1 -699.479,E2 -699.479} C_VEL
LIN {X 0,Y 601.389,Z 169.572,A -85,B 0,C 180,E1 -702.312,E2 -702.312} C_VEL
LIN {X 0,Y 601.405,Z 169.568,A -85,B 0,C 180,E1 -704.409,E2 -704.409} C_VEL
LIN {X 0,Y 601.416,Z 169.565,A -85,B 0,C 180,E1 -707.172,E2 -707.172} C_VEL
LIN {X 0,Y 601.425,Z 169.572,A -85,B 0,C 180,E1 -709.905,E2 -709.905} C_VEL
LIN {X 0,Y 601.43,Z 169.562,A -85,B 0,C 180,E1 -712.615,E2 -712.615} C_VEL
LIN {X 0,Y 601.421,Z 169.567,A -85,B 0,C 180,E1 -715.308,E2 -715.308} C_VEL
LIN {X 0,Y 601.412,Z 169.57,A -85,B 0,C 180,E1 -717.991,E2 -717.991} C_VEL
LIN {X 0,Y 601.437,Z 169.561,A -85,B 0,C 180,E1 -720.67,E2 -720.67} C_VEL
LIN {X 0,Y 601.431,Z 169.568,A -85,B 0,C 180,E1 -723.35,E2 -723.35} C_VEL
LIN {X 0,Y 601.396,Z 169.57,A -85,B 0,C 180,E1 -726.038,E2 -726.038} C_VEL
LIN {X 0,Y 601.425,Z 169.565,A -85,B 0,C 180,E1 -728.061,E2 -728.061} C_VEL
LIN {X 0,Y 601.42,Z 169.566,A -85,B 0,C 180,E1 -731.015,E2 -731.015} C_VEL
LIN {X 0,Y 601.41,Z 169.575,A -85,B 0,C 180,E1 -733.516,E2 -733.516} C_VEL
LIN {X 0,Y 601.418,Z 169.564,A -85,B 0,C 180,E1 -736.288,E2 -736.288} C_VEL
LIN {X 0,Y 601.411,Z 169.57,A -85,B 0,C 180,E1 -739.099,E2 -739.099} C_VEL
LIN {X 0,Y 601.403,Z 169.574,A -85,B 0,C 180,E1 -741.24,E2 -741.24} C_VEL
LIN {X 0,Y 601.431,Z 169.562,A -85,B 0,C 180,E1 -744.142,E2 -744.142} C_VEL
LIN {X 0,Y 601.451,Z 169.568,A -85,B 0,C 180,E1 -747.111,E2 -747.111} C_VEL
LIN {X 0,Y 601.403,Z 169.573,A -85,B 0,C 180,E1 -749.394,E2 -749.394} C_VEL
LIN {X 0,Y 601.401,Z 169.568,A -85,B 0,C 180,E1 -751.727,E2 -751.727} C_VEL
LIN {X 0,Y 601.414,Z 169.564,A -85,B 0,C 180,E1 -754.12,E2 -754.12} C_VEL
LIN {X 0,Y 601.431,Z 169.568,A -85,B 0,C 180,E1 -757.383,E2 -757.383} C_VEL
LIN {X 0,Y 601.394,Z 169.567,A -85,B 0,C 180,E1 -759.997,E2 -759.997} C_VEL
LIN {X 0,Y 601.408,Z 169.57,A -85,B 0,C 180,E1 -762.671,E2 -762.671} C_VEL
LIN {X 0,Y 601.394,Z 169.569,A -85,B 0,C 180,E1 -765.48,E2 -765.48} C_VEL
LIN {X 0,Y 601.419,Z 169.566,A -85,B 0,C 180,E1 -768.408,E2 -768.408} C_VEL
LIN {X 0,Y 601.426,Z 169.574,A -85,B 0,C 180,E1 -770.876,E2 -770.876} C_VEL
LIN {X 0,Y 601.391,Z 169.569,A -85,B 0,C 180,E1 -773.417,E2 -773.417} C_VEL
LIN {X 0,Y 601.426,Z 169.564,A -85,B 0,C 180,E1 -776.066,E2 -776.066} C_VEL
LIN {X 0,Y 601.395,Z 169.572,A -85,B 0,C 180,E1 -779.058,E2 -779.058} C_VEL
LIN {X 0,Y 601.397,Z 169.568,A -85,B 0,C 180,E1 -781.372,E2 -781.372} C_VEL
LIN {X 0,Y 601.412,Z 169.568,A -85,B 0,C 180,E1 -784.134,E2 -784.134} C_VEL
LIN {X 0,Y 601.449,Z 169.744,A -85,B 0,C 180,E1 -786.386,E2 -786.386} C_VEL
LIN {X 0,Y 601.838,Z 171.455,A -85,B 0,C 180,E1 -786.608,E2 -786.608} C_VEL
LIN {X 0,Y 601.744,Z 198.407,A -85,B 0,C 180,E1 -789.49,E2 -789.49} C_VEL
LIN {X 0,Y 601.624,Z 225.359,A -85,B 0,C 180,E1 -792.319,E2 -792.319} C_VEL
LIN {X 0,Y 601.526,Z 252.311,A -85,B 0,C 180,E1 -795.106,E2 -795.106} C_VEL
LIN {X 0,Y 601.496,Z 268.903,A -85,B 0,C 180,E1 -796.788,E2 -796.788} C_VEL
LIN {X 0,Y 601.657,Z 276.56,A -85,B 0,C 180,E1 -796.899,E2 -796.899} C_VEL
LIN {X 0,Y 601.611,Z 378.979,A -85,B 0,C 180,E1 -798.14,E2 -798.14} C_VEL
LIN {X 0,Y 601.589,Z 392.239,A -85,B 0,C 180,E1 -798.439,E2 -798.439} C_VEL
LIN {X 0,Y 601.549,Z 403.934,A -85,B 0,C 180,E1 -798.827,E2 -798.827} C_VEL
LIN {X 0,Y 601.529,Z 414.936,A -85,B 0,C 180,E1 -799.312,E2 -799.312} C_VEL
LIN {X 0,Y 601.481,Z 425.59,A -85,B 0,C 180,E1 -799.906,E2 -799.906} C_VEL
LIN {X 0,Y 601.448,Z 436.483,A -85,B 0,C 180,E1 -800.67,E2 -800.67} C_VEL
LIN {X 0,Y 601.429,Z 447.118,A -85,B 0,C 180,E1 -801.601,E2 -801.601} C_VEL
LIN {X 0,Y 601.417,Z 454.965,A -85,B 0,C 180,E1 -802.446,E2 -802.446} C_VEL
LIN {X 0,Y 601.37,Z 462.228,A -85,B 0,C 180,E1 -803.398,E2 -803.398} C_VEL
LIN {X 0,Y 601.372,Z 467.869,A -85,B 0,C 180,E1 -804.3,E2 -804.3} C_VEL
LIN {X 0,Y 601.336,Z 472.952,A -85,B 0,C 180,E1 -805.308,E2 -805.308} C_VEL
LIN {X 0,Y 601.368,Z 476.898,A -85,B 0,C 180,E1 -806.315,E2 -806.315} C_VEL
LIN {X 0,Y 601.325,Z 479.81,A -85,B 0,C 180,E1 -807.321,E2 -807.321} C_VEL
LIN {X 0,Y 601.343,Z 481.202,A -85,B 0,C 180,E1 -807.991,E2 -807.991} C_VEL
LIN {X 0,Y 601.339,Z 482.784,A -85,B 0,C 180,E1 -809.331,E2 -809.331} C_VEL
LIN {X 0,Y 601.335,Z 483,A -85,B 0,C 180,E1 -810,E2 -810} C_VEL
LIN {X 0,Y 601.347,Z 482.184,A -85,B 0,C 180,E1 -811.34,E2 -811.34} C_VEL
LIN {X 0,Y 601.343,Z 481.201,A -85,B 0,C 180,E1 -812.01,E2 -812.01} C_VEL
LIN {X 0,Y 601.325,Z 479.808,A -85,B 0,C 180,E1 -812.68,E2 -812.68} C_VEL
LIN {X 0,Y 601.368,Z 476.895,A -85,B 0,C 180,E1 -813.686,E2 -813.686} C_VEL
LIN {X 0,Y 601.336,Z 472.948,A -85,B 0,C 180,E1 -814.693,E2 -814.693} C_VEL
LIN {X 0,Y 601.372,Z 466.875,A -85,B 0,C 180,E1 -815.87,E2 -815.87} C_VEL
LIN {X 0,Y 601.382,Z 460.233,A -85,B 0,C 180,E1 -816.88,E2 -816.88} C_VEL
LIN {X 0,Y 601.4,Z 451.986,A -85,B 0,C 180,E1 -817.893,E2 -817.893} C_VEL
LIN {X 0,Y 601.436,Z 443.533,A -85,B 0,C 180,E1 -818.738,E2 -818.738} C_VEL
LIN {X 0,Y 601.449,Z 433.088,A -85,B 0,C 180,E1 -819.585,E2 -819.585} C_VEL
LIN {X 0,Y 601.476,Z 422.752,A -85,B 0,C 180,E1 -820.265,E2 -820.265} C_VEL
LIN {X 0,Y 601.538,Z 411.89,A -85,B 0,C 180,E1 -820.836,E2 -820.836} C_VEL
LIN {X 0,Y 601.566,Z 399.364,A -85,B 0,C 180,E1 -821.341,E2 -821.341} C_VEL
LIN {X 0,Y 601.605,Z 386.336,A -85,B 0,C 180,E1 -821.711,E2 -821.711} C_VEL
LIN {X 0,Y 601.622,Z 373.057,A -85,B 0,C 180,E1 -821.946,E2 -821.946} C_VEL
LIN {X 0,Y 601.565,Z 269.534,A -85,B 0,C 180,E1 -823.19,E2 -823.19} C_VEL
LIN {X 0,Y 601.508,Z 268.327,A -85,B 0,C 180,E1 -823.256,E2 -823.256} C_VEL
LIN {X 0,Y 601.578,Z 238.825,A -85,B 0,C 180,E1 -826.283,E2 -826.283} C_VEL
LIN {X 0,Y 601.652,Z 211.873,A -85,B 0,C 180,E1 -829.091,E2 -829.091} C_VEL
LIN {X 0,Y 601.782,Z 186.606,A -85,B 0,C 180,E1 -831.765,E2 -831.765} C_VEL
LIN {X 0,Y 601.846,Z 171.445,A -85,B 0,C 180,E1 -833.393,E2 -833.393} C_VEL
LIN {X 0,Y 601.435,Z 169.668,A -85,B 0,C 180,E1 -833.638,E2 -833.638} C_VEL
LIN {X 0,Y 601.386,Z 169.568,A -85,B 0,C 180,E1 -836.365,E2 -836.365} C_VEL
LIN {X 0,Y 601.405,Z 169.569,A -85,B 0,C 180,E1 -838.783,E2 -838.783} C_VEL
LIN {X 0,Y 601.42,Z 169.57,A -85,B 0,C 180,E1 -841.454,E2 -841.454} C_VEL
LIN {X 0,Y 601.41,Z 169.565,A -85,B 0,C 180,E1 -844.12,E2 -844.12} C_VEL
LIN {X 0,Y 601.394,Z 169.569,A -85,B 0,C 180,E1 -846.584,E2 -846.584} C_VEL
LIN {X 0,Y 601.414,Z 169.568,A -85,B 0,C 180,E1 -849.532,E2 -849.532} C_VEL
LIN {X 0,Y 601.413,Z 169.565,A -85,B 0,C 180,E1 -851.766,E2 -851.766} C_VEL
LIN {X 0,Y 601.4,Z 169.569,A -85,B 0,C 180,E1 -854.532,E2 -854.532} C_VEL
LIN {X 0,Y 601.411,Z 169.568,A -85,B 0,C 180,E1 -857.409,E2 -857.409} C_VEL
LIN {X 0,Y 601.4,Z 169.566,A -85,B 0,C 180,E1 -860.004,E2 -860.004} C_VEL
LIN {X 0,Y 601.436,Z 169.568,A -85,B 0,C 180,E1 -862.618,E2 -862.618} C_VEL
LIN {X 0,Y 601.419,Z 169.564,A -85,B 0,C 180,E1 -865.881,E2 -865.881} C_VEL
LIN {X 0,Y 601.418,Z 169.57,A -85,B 0,C 180,E1 -868.546,E2 -868.546} C_VEL
LIN {X 0,Y 601.429,Z 169.564,A -85,B 0,C 180,E1 -871.373,E2 -871.373} C_VEL
LIN {X 0,Y 601.393,Z 169.567,A -85,B 0,C 180,E1 -873.635,E2 -873.635} C_VEL
LIN {X 0,Y 601.415,Z 169.574,A -85,B 0,C 180,E1 -876.589,E2 -876.589} C_VEL
LIN {X 0,Y 601.421,Z 169.564,A -85,B 0,C 180,E1 -879.478,E2 -879.478} C_VEL
LIN {X 0,Y 601.39,Z 169.574,A -85,B 0,C 180,E1 -882.311,E2 -882.311} C_VEL
LIN {X 0,Y 601.407,Z 169.574,A -85,B 0,C 180,E1 -884.408,E2 -884.408} C_VEL
LIN {X 0,Y 601.413,Z 169.565,A -85,B 0,C 180,E1 -887.171,E2 -887.171} C_VEL
LIN {X 0,Y 601.424,Z 169.566,A -85,B 0,C 180,E1 -889.905,E2 -889.905} C_VEL
LIN {X 0,Y 601.441,Z 169.567,A -85,B 0,C 180,E1 -892.615,E2 -892.615} C_VEL
LIN {X 0,Y 601.408,Z 169.565,A -85,B 0,C 180,E1 -895.308,E2 -895.308} C_VEL
LIN {X 0,Y 601.419,Z 169.57,A -85,B 0,C 180,E1 -897.991,E2 -897.991} C_VEL
LIN {X 0,Y 601.438,Z 169.713,A -85,B 0,C 180,E1 -900.146,E2 -900.146} C_VEL
LIN {X 0,Y 601.474,Z 181.818,A -85,B 0,C 180,E1 -902.344,E2 -902.344} C_VEL
LIN {X 0,Y 601.44,Z 196.928,A -85,B 0,C 180,E1 -905.027,E2 -905.027} C_VEL
LIN {X 0,Y 601.385,Z 212.296,A -85,B 0,C 180,E1 -907.723,E2 -907.723} C_VEL
LIN {X 0,Y 601.418,Z 223.484,A -85,B 0,C 180,E1 -909.649,E2 -909.649} C_VEL
LIN {X 0,Y 601.506,Z 224.975,A -85,B 0,C 180,E1 -909.711,E2 -909.711} C_VEL
LIN {X 0,Y 601.523,Z 248.122,A -85,B 0,C 180,E1 -909.989,E2 -909.989} C_VEL
LIN {X 0,Y 600.84,Z 253.963,A -85,B 0,C 180,E1 -910.047,E2 -910.047} C_VEL
LIN {X 0,Y 595.155,Z 272.921,A -85,B 0,C 180,E1 -910.178,E2 -910.178} C_VEL
LIN {X 0,Y 594.509,Z 278.76,A -85,B 0,C 180,E1 -910.237,E2 -910.237} C_VEL
LIN {X 0,Y 594.53,Z 301.47,A -85,B 0,C 180,E1 -910.536,E2 -910.536} C_VEL
LIN {X 0,Y 594.491,Z 313.169,A -85,B 0,C 180,E1 -910.817,E2 -910.817} C_VEL
LIN {X 0,Y 594.45,Z 323.356,A -85,B 0,C 180,E1 -911.196,E2 -911.196} C_VEL
LIN {X 0,Y 594.424,Z 333.1,A -85,B 0,C 180,E1 -911.681,E2 -911.681} C_VEL
LIN {X 0,Y 594.38,Z 341.362,A -85,B 0,C 180,E1 -912.201,E2 -912.201} C_VEL
LIN {X 0,Y 594.35,Z 349.202,A -85,B 0,C 180,E1 -912.809,E2 -912.809} C_VEL
LIN {X 0,Y 594.303,Z 358.224,A -85,B 0,C 180,E1 -913.68,E2 -913.68} C_VEL
LIN {X 0,Y 594.294,Z 365.177,A -85,B 0,C 180,E1 -914.554,E2 -914.554} C_VEL
LIN {X 0,Y 594.295,Z 368.752,A -85,B 0,C 180,E1 -915.08,E2 -915.08} C_VEL
LIN {X 0,Y 594.272,Z 372.716,A -85,B 0,C 180,E1 -915.783,E2 -915.783} C_VEL
LIN {X 0,Y 594.251,Z 376.69,A -85,B 0,C 180,E1 -916.673,E2 -916.673} C_VEL
LIN {X 0,Y 594.211,Z 380.439,A -85,B 0,C 180,E1 -917.909,E2 -917.909} C_VEL
LIN {X 0,Y 594.235,Z 382.21,A -85,B 0,C 180,E1 -918.888,E2 -918.888} C_VEL
LIN {X 0,Y 594.214,Z 382.999,A -85,B 0,C 180,E1 -920.059,E2 -920.059} C_VEL
LIN {X 0,Y 594.247,Z 382.62,A -85,B 0,C 180,E1 -920.883,E2 -920.883} C_VEL
LIN {X 0,Y 594.226,Z 381.786,A -85,B 0,C 180,E1 -921.508,E2 -921.508} C_VEL
LIN {X 0,Y 594.254,Z 379.091,A -85,B 0,C 180,E1 -922.71,E2 -922.71} C_VEL
LIN {X 0,Y 594.247,Z 375.437,A -85,B 0,C 180,E1 -923.71,E2 -923.71} C_VEL
LIN {X 0,Y 594.281,Z 370.87,A -85,B 0,C 180,E1 -924.637,E2 -924.637} C_VEL
LIN {X 0,Y 594.288,Z 366.228,A -85,B 0,C 180,E1 -925.384,E2 -925.384} C_VEL
LIN {X 0,Y 594.327,Z 360.681,A -85,B 0,C 180,E1 -926.115,E2 -926.115} C_VEL
LIN {X 0,Y 594.322,Z 355.383,A -85,B 0,C 180,E1 -926.702,E2 -926.702} C_VEL
LIN {X 0,Y 594.329,Z 348.179,A -85,B 0,C 180,E1 -927.367,E2 -927.367} C_VEL
LIN {X 0,Y 594.369,Z 339.546,A -85,B 0,C 180,E1 -928.016,E2 -928.016} C_VEL
LIN {X 0,Y 594.43,Z 328.508,A -85,B 0,C 180,E1 -928.657,E2 -928.657} C_VEL
LIN {X 0,Y 594.474,Z 318.383,A -85,B 0,C 180,E1 -929.09,E2 -929.09} C_VEL
LIN {X 0,Y 594.486,Z 308.715,A -85,B 0,C 180,E1 -929.393,E2 -929.393} C_VEL
LIN {X 0,Y 594.52,Z 299.597,A -85,B 0,C 180,E1 -929.585,E2 -929.585} C_VEL
LIN {X 0,Y 594.402,Z 224.172,A -85,B 0,C 180,E1 -930.52,E2 -930.52} C_VEL
LIN {X 0,Y 594.35,Z 222.841,A -85,B 0,C 180,E1 -930.659,E2 -930.659} C_VEL
LIN {X 0,Y 594.357,Z 206.401,A -85,B 0,C 180,E1 -933.559,E2 -933.559} C_VEL
LIN {X 0,Y 594.414,Z 191.373,A -85,B 0,C 180,E1 -936.24,E2 -936.24} C_VEL
LIN {X 0,Y 594.516,Z 176.037,A -85,B 0,C 180,E1 -939.012,E2 -939.012} C_VEL
LIN {X 0,Y 594.418,Z 170.556,A -85,B 0,C 180,E1 -940.042,E2 -940.042} C_VEL
LIN {X 0,Y 594.357,Z 170.444,A -85,B 0,C 180,E1 -942.851,E2 -942.851} C_VEL
LIN {X 0,Y 594.376,Z 170.452,A -85,B 0,C 180,E1 -945.763,E2 -945.763} C_VEL
LIN {X 0,Y 594.379,Z 170.441,A -85,B 0,C 180,E1 -948.536,E2 -948.536} C_VEL
LIN {X 0,Y 594.378,Z 170.445,A -85,B 0,C 180,E1 -951.296,E2 -951.296} C_VEL
LIN {X 0,Y 594.392,Z 170.447,A -85,B 0,C 180,E1 -953.758,E2 -953.758} C_VEL
LIN {X 0,Y 594.377,Z 170.442,A -85,B 0,C 180,E1 -956.239,E2 -956.239} C_VEL
LIN {X 0,Y 594.367,Z 170.442,A -85,B 0,C 180,E1 -958.649,E2 -958.649} C_VEL
LIN {X 0,Y 594.382,Z 170.443,A -85,B 0,C 180,E1 -961.042,E2 -961.042} C_VEL
LIN {X 0,Y 594.379,Z 170.442,A -85,B 0,C 180,E1 -964.056,E2 -964.056} C_VEL
LIN {X 0,Y 594.389,Z 170.44,A -85,B 0,C 180,E1 -966.296,E2 -966.296} C_VEL
LIN {X 0,Y 594.403,Z 170.445,A -85,B 0,C 180,E1 -969.224,E2 -969.224} C_VEL
LIN {X 0,Y 594.352,Z 170.445,A -85,B 0,C 180,E1 -972.095,E2 -972.095} C_VEL
LIN {X 0,Y 594.363,Z 170.443,A -85,B 0,C 180,E1 -974.219,E2 -974.219} C_VEL
LIN {X 0,Y 594.379,Z 170.441,A -85,B 0,C 180,E1 -976.321,E2 -976.321} C_VEL
LIN {X 0,Y 594.378,Z 170.448,A -85,B 0,C 180,E1 -979.094,E2 -979.094} C_VEL
LIN {X 0,Y 594.416,Z 170.437,A -85,B 0,C 180,E1 -981.843,E2 -981.843} C_VEL
LIN {X 0,Y 594.391,Z 170.441,A -85,B 0,C 180,E1 -984.572,E2 -984.572} C_VEL
LIN {X 0,Y 594.405,Z 170.445,A -85,B 0,C 180,E1 -987.289,E2 -987.289} C_VEL
LIN {X 0,Y 594.414,Z 170.436,A -85,B 0,C 180,E1 -990,E2 -990} C_VEL
LIN {X 0,Y 594.4,Z 170.443,A -85,B 0,C 180,E1 -992.71,E2 -992.71} C_VEL
LIN {X 0,Y 594.395,Z 170.442,A -85,B 0,C 180,E1 -995.427,E2 -995.427} C_VEL
LIN {X 0,Y 594.411,Z 170.437,A -85,B 0,C 180,E1 -998.156,E2 -998.156} C_VEL
LIN {X 0,Y 594.388,Z 170.447,A -85,B 0,C 180,E1 -1001.074,E2 -1001.074} C_VEL
LIN {X 0,Y 594.381,Z 170.441,A -85,B 0,C 180,E1 -1003.678,E2 -1003.678} C_VEL
LIN {X 0,Y 594.389,Z 170.448,A -85,B 0,C 180,E1 -1006.719,E2 -1006.719} C_VEL
LIN {X 0,Y 594.363,Z 170.445,A -85,B 0,C 180,E1 -1009.334,E2 -1009.334} C_VEL
LIN {X 0,Y 594.363,Z 170.443,A -85,B 0,C 180,E1 -1011.503,E2 -1011.503} C_VEL
LIN {X 0,Y 594.383,Z 170.446,A -85,B 0,C 180,E1 -1014.446,E2 -1014.446} C_VEL
LIN {X 0,Y 594.381,Z 170.45,A -85,B 0,C 180,E1 -1016.699,E2 -1016.699} C_VEL
LIN {X 0,Y 594.378,Z 170.445,A -85,B 0,C 180,E1 -1018.998,E2 -1018.998} C_VEL
LIN {X 0,Y 594.387,Z 170.44,A -85,B 0,C 180,E1 -1021.645,E2 -1021.645} C_VEL
LIN {X 0,Y 594.39,Z 170.449,A -85,B 0,C 180,E1 -1024.578,E2 -1024.578} C_VEL
LIN {X 0,Y 594.378,Z 170.442,A -85,B 0,C 180,E1 -1027.086,E2 -1027.086} C_VEL
LIN {X 0,Y 594.37,Z 170.443,A -85,B 0,C 180,E1 -1029.774,E2 -1029.774} C_VEL
LIN {X 0,Y 594.366,Z 170.452,A -85,B 0,C 180,E1 -1032.374,E2 -1032.374} C_VEL
LIN {X 0,Y 594.355,Z 170.444,A -85,B 0,C 180,E1 -1035.191,E2 -1035.191} C_VEL
LIN {X 0,Y 594.377,Z 170.448,A -85,B 0,C 180,E1 -1038.151,E2 -1038.151} C_VEL
LIN {X 0,Y 594.388,Z 170.45,A -85,B 0,C 180,E1 -1040.321,E2 -1040.321} C_VEL
LIN {X 0,Y 594.377,Z 170.442,A -85,B 0,C 180,E1 -1042.913,E2 -1042.913} C_VEL
LIN {X 0,Y 594.379,Z 170.445,A -85,B 0,C 180,E1 -1045.86,E2 -1045.86} C_VEL
LIN {X 0,Y 594.382,Z 170.443,A -85,B 0,C 180,E1 -1048.651,E2 -1048.651} C_VEL
LIN {X 0,Y 594.379,Z 170.441,A -85,B 0,C 180,E1 -1051.041,E2 -1051.041} C_VEL
LIN {X 0,Y 594.381,Z 170.449,A -85,B 0,C 180,E1 -1053.976,E2 -1053.976} C_VEL
LIN {X 0,Y 594.388,Z 170.446,A -85,B 0,C 180,E1 -1056.296,E2 -1056.296} C_VEL
LIN {X 0,Y 594.401,Z 170.438,A -85,B 0,C 180,E1 -1059.225,E2 -1059.225} C_VEL
LIN {X 0,Y 594.373,Z 170.449,A -85,B 0,C 180,E1 -1062.096,E2 -1062.096} C_VEL
LIN {X 0,Y 594.36,Z 170.448,A -85,B 0,C 180,E1 -1064.219,E2 -1064.219} C_VEL
LIN {X 0,Y 594.361,Z 170.443,A -85,B 0,C 180,E1 -1067.017,E2 -1067.017} C_VEL
LIN {X 0,Y 594.386,Z 170.449,A -85,B 0,C 180,E1 -1069.784,E2 -1069.784} C_VEL
LIN {X 0,Y 594.384,Z 170.441,A -85,B 0,C 180,E1 -1072.527,E2 -1072.527} C_VEL
LIN {X 0,Y 594.389,Z 170.442,A -85,B 0,C 180,E1 -1075.253,E2 -1075.253} C_VEL
LIN {X 0,Y 594.383,Z 170.446,A -85,B 0,C 180,E1 -1077.968,E2 -1077.968} C_VEL
LIN {X 0,Y 594.409,Z 170.437,A -85,B 0,C 180,E1 -1080.678,E2 -1080.678} C_VEL
LIN {X 0,Y 594.382,Z 170.447,A -85,B 0,C 180,E1 -1083.39,E2 -1083.39} C_VEL
LIN {X 0,Y 594.35,Z 170.446,A -85,B 0,C 180,E1 -1086.109,E2 -1086.109} C_VEL
LIN {X 0,Y 594.371,Z 170.443,A -85,B 0,C 180,E1 -1088.158,E2 -1088.158} C_VEL
LIN {X 0,Y 594.383,Z 170.444,A -85,B 0,C 180,E1 -1091.076,E2 -1091.076} C_VEL
LIN {X 0,Y 594.368,Z 170.449,A -85,B 0,C 180,E1 -1093.68,E2 -1093.68} C_VEL
LIN {X 0,Y 594.381,Z 170.441,A -85,B 0,C 180,E1 -1096.718,E2 -1096.718} C_VEL
LIN {X 0,Y 594.359,Z 170.453,A -85,B 0,C 180,E1 -1099.335,E2 -1099.335} C_VEL
LIN {X 0,Y 594.359,Z 170.451,A -85,B 0,C 180,E1 -1101.504,E2 -1101.504} C_VEL
LIN {X 0,Y 594.381,Z 170.441,A -85,B 0,C 180,E1 -1104.447,E2 -1104.447} C_VEL
LIN {X 0,Y 594.368,Z 170.449,A -85,B 0,C 180,E1 -1107.462,E2 -1107.462} C_VEL
LIN {X 0,Y 594.363,Z 170.443,A -85,B 0,C 180,E1 -1110.326,E2 -1110.326} C_VEL
LIN {X 0,Y 594.371,Z 170.448,A -85,B 0,C 180,E1 -1112.951,E2 -1112.951} C_VEL
LIN {X 0,Y 594.343,Z 170.451,A -85,B 0,C 180,E1 -1115.41,E2 -1115.41} C_VEL
LIN {X 0,Y 594.372,Z 170.442,A -85,B 0,C 180,E1 -1117.942,E2 -1117.942} C_VEL
LIN {X 0,Y 594.371,Z 170.448,A -85,B 0,C 180,E1 -1120.823,E2 -1120.823} C_VEL
LIN {X 0,Y 594.347,Z 170.45,A -85,B 0,C 180,E1 -1123.302,E2 -1123.302} C_VEL
LIN {X 0,Y 594.356,Z 170.444,A -85,B 0,C 180,E1 -1126.162,E2 -1126.162} C_VEL
LIN {X 0,Y 594.371,Z 170.447,A -85,B 0,C 180,E1 -1129.179,E2 -1129.179} C_VEL
LIN {X 0,Y 594.37,Z 170.442,A -85,B 0,C 180,E1 -1132.059,E2 -1132.059} C_VEL
LIN {X 0,Y 594.347,Z 170.453,A -85,B 0,C 180,E1 -1134.678,E2 -1134.678} C_VEL
LIN {X 0,Y 594.37,Z 170.447,A -85,B 0,C 180,E1 -1137.09,E2 -1137.09} C_VEL
LIN {X 0,Y 594.364,Z 170.443,A -85,B 0,C 180,E1 -1139.676,E2 -1139.676} C_VEL
LIN {X 0,Y 594.374,Z 170.45,A -85,B 0,C 180,E1 -1142.54,E2 -1142.54} C_VEL
LIN {X 0,Y 594.37,Z 170.45,A -85,B 0,C 180,E1 -1144.807,E2 -1144.807} C_VEL
LIN {X 0,Y 594.418,Z 170.605,A -85,B 0,C 180,E1 -1146.182,E2 -1146.182} C_VEL
LIN {X 0,Y 595.003,Z 173.139,A -85,B 0,C 180,E1 -1146.507,E2 -1146.507} C_VEL
LIN {X 0,Y 594.856,Z 198.407,A -85,B 0,C 180,E1 -1149.242,E2 -1149.242} C_VEL
LIN {X 0,Y 594.685,Z 225.359,A -85,B 0,C 180,E1 -1152.106,E2 -1152.106} C_VEL
LIN {X 0,Y 594.561,Z 250.626,A -85,B 0,C 180,E1 -1154.752,E2 -1154.752} C_VEL
LIN {X 0,Y 594.503,Z 268.901,A -85,B 0,C 180,E1 -1156.629,E2 -1156.629} C_VEL
LIN {X 0,Y 594.74,Z 274.771,A -85,B 0,C 180,E1 -1156.722,E2 -1156.722} C_VEL
LIN {X 0,Y 594.663,Z 378.979,A -85,B 0,C 180,E1 -1157.999,E2 -1157.999} C_VEL
LIN {X 0,Y 594.637,Z 392.239,A -85,B 0,C 180,E1 -1158.302,E2 -1158.302} C_VEL
LIN {X 0,Y 594.595,Z 404.58,A -85,B 0,C 180,E1 -1158.719,E2 -1158.719} C_VEL
LIN {X 0,Y 594.537,Z 416.643,A -85,B 0,C 180,E1 -1159.271,E2 -1159.271} C_VEL
LIN {X 0,Y 594.482,Z 428.209,A -85,B 0,C 180,E1 -1159.958,E2 -1159.958} C_VEL
LIN {X 0,Y 594.414,Z 438.604,A -85,B 0,C 180,E1 -1160.73,E2 -1160.73} C_VEL
LIN {X 0,Y 594.383,Z 447.118,A -85,B 0,C 180,E1 -1161.501,E2 -1161.501} C_VEL
LIN {X 0,Y 594.347,Z 454.965,A -85,B 0,C 180,E1 -1162.356,E2 -1162.356} C_VEL
LIN {X 0,Y 594.282,Z 462.816,A -85,B 0,C 180,E1 -1163.409,E2 -1163.409} C_VEL
LIN {X 0,Y 594.289,Z 469.683,A -85,B 0,C 180,E1 -1164.572,E2 -1164.572} C_VEL
LIN {X 0,Y 594.27,Z 474.374,A -85,B 0,C 180,E1 -1165.592,E2 -1165.592} C_VEL
LIN {X 0,Y 594.267,Z 477.958,A -85,B 0,C 180,E1 -1166.611,E2 -1166.611} C_VEL
LIN {X 0,Y 594.226,Z 479.81,A -85,B 0,C 180,E1 -1167.289,E2 -1167.289} C_VEL
LIN {X 0,Y 594.242,Z 481.202,A -85,B 0,C 180,E1 -1167.967,E2 -1167.967} C_VEL
LIN {X 0,Y 594.239,Z 482.784,A -85,B 0,C 180,E1 -1169.323,E2 -1169.323} C_VEL
LIN {X 0,Y 594.236,Z 483,A -85,B 0,C 180,E1 -1170,E2 -1170} C_VEL
LIN {X 0,Y 594.247,Z 482.184,A -85,B 0,C 180,E1 -1171.356,E2 -1171.356} C_VEL
LIN {X 0,Y 594.242,Z 481.201,A -85,B 0,C 180,E1 -1172.034,E2 -1172.034} C_VEL
LIN {X 0,Y 594.226,Z 479.808,A -85,B 0,C 180,E1 -1172.712,E2 -1172.712} C_VEL
LIN {X 0,Y 594.289,Z 476.895,A -85,B 0,C 180,E1 -1173.73,E2 -1173.73} C_VEL
LIN {X 0,Y 594.241,Z 472.948,A -85,B 0,C 180,E1 -1174.749,E2 -1174.749} C_VEL
LIN {X 0,Y 594.304,Z 466.875,A -85,B 0,C 180,E1 -1175.94,E2 -1175.94} C_VEL
LIN {X 0,Y 594.308,Z 460.233,A -85,B 0,C 180,E1 -1176.962,E2 -1176.962} C_VEL
LIN {X 0,Y 594.359,Z 451.986,A -85,B 0,C 180,E1 -1177.987,E2 -1177.987} C_VEL
LIN {X 0,Y 594.382,Z 443.533,A -85,B 0,C 180,E1 -1178.843,E2 -1178.843} C_VEL
LIN {X 0,Y 594.434,Z 433.089,A -85,B 0,C 180,E1 -1179.7,E2 -1179.7} C_VEL
LIN {X 0,Y 594.491,Z 422.752,A -85,B 0,C 180,E1 -1180.387,E2 -1180.387} C_VEL
LIN {X 0,Y 594.562,Z 411.684,A -85,B 0,C 180,E1 -1180.975,E2 -1180.975} C_VEL
LIN {X 0,Y 594.601,Z 399.69,A -85,B 0,C 180,E1 -1181.464,E2 -1181.464} C_VEL
LIN {X 0,Y 594.647,Z 386.335,A -85,B 0,C 180,E1 -1181.85,E2 -1181.85} C_VEL
LIN {X 0,Y 594.695,Z 373.057,A -85,B 0,C 180,E1 -1182.087,E2 -1182.087} C_VEL
LIN {X 0,Y 594.597,Z 269.534,A -85,B 0,C 180,E1 -1183.348,E2 -1183.348} C_VEL
LIN {X 0,Y 594.475,Z 268.327,A -85,B 0,C 180,E1 -1183.416,E2 -1183.416} C_VEL
LIN {X 0,Y 594.629,Z 240.51,A -85,B 0,C 180,E1 -1186.303,E2 -1186.303} C_VEL
LIN {X 0,Y 594.763,Z 211.873,A -85,B 0,C 180,E1 -1189.321,E2 -1189.321} C_VEL
LIN {X 0,Y 594.946,Z 186.606,A -85,B 0,C 180,E1 -1192.028,E2 -1192.028} C_VEL
LIN {X 0,Y 594.997,Z 173.13,A -85,B 0,C 180,E1 -1193.494,E2 -1193.494} C_VEL
LIN {X 0,Y 594.402,Z 170.526,A -85,B 0,C 180,E1 -1193.843,E2 -1193.843} C_VEL
LIN {X 0,Y 594.365,Z 170.445,A -85,B 0,C 180,E1 -1196.701,E2 -1196.701} C_VEL
LIN {X 0,Y 594.373,Z 170.448,A -85,B 0,C 180,E1 -1198.999,E2 -1198.999} C_VEL
LIN {X 0,Y 594.374,Z 170.445,A -85,B 0,C 180,E1 -1201.642,E2 -1201.642} C_VEL
LIN {X 0,Y 594.367,Z 170.444,A -85,B 0,C 180,E1 -1204.581,E2 -1204.581} C_VEL
LIN {X 0,Y 594.387,Z 170.443,A -85,B 0,C 180,E1 -1207.608,E2 -1207.608} C_VEL
LIN {X 0,Y 594.362,Z 170.446,A -85,B 0,C 180,E1 -1210.568,E2 -1210.568} C_VEL
LIN {X 0,Y 594.361,Z 170.449,A -85,B 0,C 180,E1 -1213.3,E2 -1213.3} C_VEL
LIN {X 0,Y 594.345,Z 170.445,A -85,B 0,C 180,E1 -1216.163,E2 -1216.163} C_VEL
LIN {X 0,Y 594.372,Z 170.445,A -85,B 0,C 180,E1 -1218.535,E2 -1218.535} C_VEL
LIN {X 0,Y 594.372,Z 170.445,A -85,B 0,C 180,E1 -1221.297,E2 -1221.297} C_VEL
LIN {X 0,Y 594.348,Z 170.445,A -85,B 0,C 180,E1 -1223.755,E2 -1223.755} C_VEL
LIN {X 0,Y 594.365,Z 170.444,A -85,B 0,C 180,E1 -1226.238,E2 -1226.238} C_VEL
LIN {X 0,Y 594.367,Z 170.451,A -85,B 0,C 180,E1 -1228.649,E2 -1228.649} C_VEL
LIN {X 0,Y 594.383,Z 170.445,A -85,B 0,C 180,E1 -1231.042,E2 -1231.042} C_VEL
LIN {X 0,Y 594.374,Z 170.442,A -85,B 0,C 180,E1 -1233.98,E2 -1233.98} C_VEL
LIN {X 0,Y 594.379,Z 170.445,A -85,B 0,C 180,E1 -1236.295,E2 -1236.295} C_VEL
LIN {X 0,Y 594.401,Z 170.439,A -85,B 0,C 180,E1 -1239.224,E2 -1239.224} C_VEL
LIN {X 0,Y 594.342,Z 170.449,A -85,B 0,C 180,E1 -1242.094,E2 -1242.094} C_VEL
LIN {X 0,Y 594.358,Z 170.449,A -85,B 0,C 180,E1 -1244.219,E2 -1244.219} C_VEL
LIN {X 0,Y 594.37,Z 170.45,A -85,B 0,C 180,E1 -1246.32,E2 -1246.32} C_VEL
LIN {X 0,Y 594.373,Z 170.443,A -85,B 0,C 180,E1 -1249.094,E2 -1249.094} C_VEL
LIN {X 0,Y 594.378,Z 170.443,A -85,B 0,C 180,E1 -1251.842,E2 -1251.842} C_VEL
LIN {X 0,Y 594.392,Z 170.446,A -85,B 0,C 180,E1 -1254.572,E2 -1254.572} C_VEL
LIN {X 0,Y 594.399,Z 170.439,A -85,B 0,C 180,E1 -1257.289,E2 -1257.289} C_VEL
LIN {X 0,Y 594.409,Z 170.594,A -85,B 0,C 180,E1 -1260.063,E2 -1260.063} C_VEL
LIN {X 0,Y 594.457,Z 183.163,A -85,B 0,C 180,E1 -1262.371,E2 -1262.371} C_VEL
LIN {X 0,Y 594.414,Z 198.279,A -85,B 0,C 180,E1 -1265.087,E2 -1265.087} C_VEL
LIN {X 0,Y 594.332,Z 213.659,A -85,B 0,C 180,E1 -1267.815,E2 -1267.815} C_VEL
LIN {X 0,Y 594.346,Z 223.54,A -85,B 0,C 180,E1 -1269.529,E2 -1269.529} C_VEL
LIN {X 0,Y 594.51,Z 225.096,A -85,B 0,C 180,E1 -1269.59,E2 -1269.59} C_VEL
LIN {X 0,Y 594.509,Z 278.76,A -85,B 0,C 180,E1 -1270.237,E2 -1270.237} C_VEL
LIN {X 0,Y 593.833,Z 282.681,A -85,B 0,C 180,E1 -1270.272,E2 -1270.272} C_VEL
LIN {X 0,Y 588.146,Z 294.942,A -85,B 0,C 180,E1 -1270.326,E2 -1270.326} C_VEL
LIN {X 0,Y 587.541,Z 298.835,A -85,B 0,C 180,E1 -1270.378,E2 -1270.378} C_VEL
LIN {X 0,Y 587.496,Z 307.538,A -85,B 0,C 180,E1 -1270.555,E2 -1270.555} C_VEL
LIN {X 0,Y 587.479,Z 316.3,A -85,B 0,C 180,E1 -1270.816,E2 -1270.816} C_VEL
LIN {X 0,Y 587.436,Z 325.243,A -85,B 0,C 180,E1 -1271.177,E2 -1271.177} C_VEL
LIN {X 0,Y 587.375,Z 334.125,A -85,B 0,C 180,E1 -1271.64,E2 -1271.64} C_VEL
LIN {X 0,Y 587.334,Z 343.556,A -85,B 0,C 180,E1 -1272.262,E2 -1272.262} C_VEL
LIN {X 0,Y 587.284,Z 352.002,A -85,B 0,C 180,E1 -1272.966,E2 -1272.966} C_VEL
LIN {X 0,Y 587.239,Z 358.795,A -85,B 0,C 180,E1 -1273.672,E2 -1273.672} C_VEL
LIN {X 0,Y 587.23,Z 363.951,A -85,B 0,C 180,E1 -1274.309,E2 -1274.309} C_VEL
LIN {X 0,Y 587.188,Z 370.14,A -85,B 0,C 180,E1 -1275.267,E2 -1275.267} C_VEL
LIN {X 0,Y 587.162,Z 375.438,A -85,B 0,C 180,E1 -1276.336,E2 -1276.336} C_VEL
LIN {X 0,Y 587.139,Z 379.292,A -85,B 0,C 180,E1 -1277.412,E2 -1277.412} C_VEL
LIN {X 0,Y 587.128,Z 381.022,A -85,B 0,C 180,E1 -1278.133,E2 -1278.133} C_VEL
LIN {X 0,Y 587.144,Z 382.362,A -85,B 0,C 180,E1 -1278.984,E2 -1278.984} C_VEL
LIN {X 0,Y 587.109,Z 382.814,A -85,B 0,C 180,E1 -1279.583,E2 -1279.583} C_VEL
LIN {X 0,Y 587.118,Z 382.903,A -85,B 0,C 180,E1 -1280.312,E2 -1280.312} C_VEL
LIN {X 0,Y 587.143,Z 382.447,A -85,B 0,C 180,E1 -1281.044,E2 -1281.044} C_VEL
LIN {X 0,Y 587.143,Z 381.405,A -85,B 0,C 180,E1 -1281.781,E2 -1281.781} C_VEL
LIN {X 0,Y 587.151,Z 378.8,A -85,B 0,C 180,E1 -1282.83,E2 -1282.83} C_VEL
LIN {X 0,Y 587.167,Z 375.947,A -85,B 0,C 180,E1 -1283.639,E2 -1283.639} C_VEL
LIN {X 0,Y 587.199,Z 371.676,A -85,B 0,C 180,E1 -1284.547,E2 -1284.547} C_VEL
LIN {X 0,Y 587.217,Z 367.025,A -85,B 0,C 180,E1 -1285.332,E2 -1285.332} C_VEL
LIN {X 0,Y 587.243,Z 360.937,A -85,B 0,C 180,E1 -1286.158,E2 -1286.158} C_VEL
LIN {X 0,Y 587.264,Z 354.653,A -85,B 0,C 180,E1 -1286.857,E2 -1286.857} C_VEL
LIN {X 0,Y 587.314,Z 347.354,A -85,B 0,C 180,E1 -1287.525,E2 -1287.525} C_VEL
LIN {X 0,Y 587.366,Z 338.211,A -85,B 0,C 180,E1 -1288.205,E2 -1288.205} C_VEL
LIN {X 0,Y 587.426,Z 328.442,A -85,B 0,C 180,E1 -1288.764,E2 -1288.764} C_VEL
LIN {X 0,Y 587.464,Z 319.648,A -85,B 0,C 180,E1 -1289.153,E2 -1289.153} C_VEL
LIN {X 0,Y 587.501,Z 309.611,A -85,B 0,C 180,E1 -1289.481,E2 -1289.481} C_VEL
LIN {X 0,Y 587.513,Z 300.201,A -85,B 0,C 180,E1 -1289.69,E2 -1289.69} C_VEL
LIN {X 0,Y 587.49,Z 225.42,A -85,B 0,C 180,E1 -1290.62,E2 -1290.62} C_VEL
LIN {X 0,Y 587.302,Z 223.55,A -85,B 0,C 180,E1 -1290.689,E2 -1290.689} C_VEL
LIN {X 0,Y 587.339,Z 208.224,A -85,B 0,C 180,E1 -1293.396,E2 -1293.396} C_VEL
LIN {X 0,Y 587.397,Z 193.242,A -85,B 0,C 180,E1 -1296.099,E2 -1296.099} C_VEL
LIN {X 0,Y 587.518,Z 177.568,A -85,B 0,C 180,E1 -1298.964,E2 -1298.964} C_VEL
LIN {X 0,Y 587.382,Z 171.393,A -85,B 0,C 180,E1 -1300.143,E2 -1300.143} C_VEL
LIN {X 0,Y 587.312,Z 171.322,A -85,B 0,C 180,E1 -1303.118,E2 -1303.118} C_VEL
LIN {X 0,Y 587.322,Z 171.326,A -85,B 0,C 180,E1 -1306.049,E2 -1306.049} C_VEL
LIN {X 0,Y 587.333,Z 171.319,A -85,B 0,C 180,E1 -1308.925,E2 -1308.925} C_VEL
LIN {X 0,Y 587.325,Z 171.327,A -85,B 0,C 180,E1 -1311.52,E2 -1311.52} C_VEL
LIN {X 0,Y 587.316,Z 171.323,A -85,B 0,C 180,E1 -1314.102,E2 -1314.102} C_VEL
LIN {X 0,Y 587.339,Z 171.318,A -85,B 0,C 180,E1 -1316.888,E2 -1316.888} C_VEL
LIN {X 0,Y 587.332,Z 171.324,A -85,B 0,C 180,E1 -1319.83,E2 -1319.83} C_VEL
LIN {X 0,Y 587.34,Z 171.318,A -85,B 0,C 180,E1 -1322.308,E2 -1322.308} C_VEL
LIN {X 0,Y 587.336,Z 171.318,A -85,B 0,C 180,E1 -1324.483,E2 -1324.483} C_VEL
LIN {X 0,Y 587.317,Z 171.326,A -85,B 0,C 180,E1 -1327.131,E2 -1327.131} C_VEL
LIN {X 0,Y 587.328,Z 171.324,A -85,B 0,C 180,E1 -1329.695,E2 -1329.695} C_VEL
LIN {X 0,Y 587.348,Z 171.317,A -85,B 0,C 180,E1 -1332.594,E2 -1332.594} C_VEL
LIN {X 0,Y 587.364,Z 171.318,A -85,B 0,C 180,E1 -1335.739,E2 -1335.739} C_VEL
LIN {X 0,Y 587.346,Z 171.321,A -85,B 0,C 180,E1 -1338.866,E2 -1338.866} C_VEL
LIN {X 0,Y 587.369,Z 171.316,A -85,B 0,C 180,E1 -1341.744,E2 -1341.744} C_VEL
LIN {X 0,Y 587.358,Z 171.316,A -85,B 0,C 180,E1 -1344.507,E2 -1344.507} C_VEL
LIN {X 0,Y 587.371,Z 171.322,A -85,B 0,C 180,E1 -1347.256,E2 -1347.256} C_VEL
LIN {X 0,Y 587.382,Z 171.312,A -85,B 0,C 180,E1 -1350,E2 -1350} C_VEL
LIN {X 0,Y 587.367,Z 171.319,A -85,B 0,C 180,E1 -1352.743,E2 -1352.743} C_VEL
LIN {X 0,Y 587.361,Z 171.317,A -85,B 0,C 180,E1 -1355.492,E2 -1355.492} C_VEL
LIN {X 0,Y 587.363,Z 171.316,A -85,B 0,C 180,E1 -1358.255,E2 -1358.255} C_VEL
LIN {X 0,Y 587.345,Z 171.323,A -85,B 0,C 180,E1 -1361.133,E2 -1361.133} C_VEL
LIN {X 0,Y 587.362,Z 171.316,A -85,B 0,C 180,E1 -1364.26,E2 -1364.26} C_VEL
LIN {X 0,Y 587.347,Z 171.318,A -85,B 0,C 180,E1 -1367.405,E2 -1367.405} C_VEL
LIN {X 0,Y 587.326,Z 171.322,A -85,B 0,C 180,E1 -1370.304,E2 -1370.304} C_VEL
LIN {X 0,Y 587.319,Z 171.322,A -85,B 0,C 180,E1 -1373.258,E2 -1373.258} C_VEL
LIN {X 0,Y 587.335,Z 171.318,A -85,B 0,C 180,E1 -1375.516,E2 -1375.516} C_VEL
LIN {X 0,Y 587.344,Z 171.317,A -85,B 0,C 180,E1 -1377.817,E2 -1377.817} C_VEL
LIN {X 0,Y 587.336,Z 171.327,A -85,B 0,C 180,E1 -1380.51,E2 -1380.51} C_VEL
LIN {X 0,Y 587.335,Z 171.32,A -85,B 0,C 180,E1 -1383.112,E2 -1383.112} C_VEL
LIN {X 0,Y 587.351,Z 171.318,A -85,B 0,C 180,E1 -1385.895,E2 -1385.895} C_VEL
LIN {X 0,Y 587.325,Z 171.33,A -85,B 0,C 180,E1 -1388.479,E2 -1388.479} C_VEL
LIN {X 0,Y 587.33,Z 171.319,A -85,B 0,C 180,E1 -1391.156,E2 -1391.156} C_VEL
LIN {X 0,Y 587.326,Z 171.325,A -85,B 0,C 180,E1 -1394.114,E2 -1394.114} C_VEL
LIN {X 0,Y 587.307,Z 171.323,A -85,B 0,C 180,E1 -1396.993,E2 -1396.993} C_VEL
LIN {X 0,Y 587.321,Z 171.322,A -85,B 0,C 180,E1 -1399.747,E2 -1399.747} C_VEL
LIN {X 0,Y 587.337,Z 171.326,A -85,B 0,C 180,E1 -1402.392,E2 -1402.392} C_VEL
LIN {X 0,Y 587.341,Z 171.318,A -85,B 0,C 180,E1 -1404.946,E2 -1404.946} C_VEL
LIN {X 0,Y 587.334,Z 171.319,A -85,B 0,C 180,E1 -1407.421,E2 -1407.421} C_VEL
LIN {X 0,Y 587.339,Z 171.323,A -85,B 0,C 180,E1 -1409.831,E2 -1409.831} C_VEL
LIN {X 0,Y 587.343,Z 171.324,A -85,B 0,C 180,E1 -1412.307,E2 -1412.307} C_VEL
LIN {X 0,Y 587.328,Z 171.323,A -85,B 0,C 180,E1 -1414.483,E2 -1414.483} C_VEL
LIN {X 0,Y 587.312,Z 171.321,A -85,B 0,C 180,E1 -1417.131,E2 -1417.131} C_VEL
LIN {X 0,Y 587.325,Z 171.325,A -85,B 0,C 180,E1 -1419.695,E2 -1419.695} C_VEL
LIN {X 0,Y 587.349,Z 171.318,A -85,B 0,C 180,E1 -1422.594,E2 -1422.594} C_VEL
LIN {X 0,Y 587.356,Z 171.323,A -85,B 0,C 180,E1 -1425.739,E2 -1425.739} C_VEL
LIN {X 0,Y 587.354,Z 171.316,A -85,B 0,C 180,E1 -1428.859,E2 -1428.859} C_VEL
LIN {X 0,Y 587.361,Z 171.324,A -85,B 0,C 180,E1 -1431.745,E2 -1431.745} C_VEL
LIN {X 0,Y 587.346,Z 171.317,A -85,B 0,C 180,E1 -1434.507,E2 -1434.507} C_VEL
LIN {X 0,Y 587.371,Z 171.317,A -85,B 0,C 180,E1 -1437.257,E2 -1437.257} C_VEL
LIN {X 0,Y 587.37,Z 171.319,A -85,B 0,C 180,E1 -1440,E2 -1440} C_VEL
LIN {X 0,Y 587.362,Z 171.315,A -85,B 0,C 180,E1 -1442.744,E2 -1442.744} C_VEL
LIN {X 0,Y 587.353,Z 171.325,A -85,B 0,C 180,E1 -1445.493,E2 -1445.493} C_VEL
LIN {X 0,Y 587.332,Z 171.319,A -85,B 0,C 180,E1 -1448.256,E2 -1448.256} C_VEL
LIN {X 0,Y 587.34,Z 171.322,A -85,B 0,C 180,E1 -1451.134,E2 -1451.134} C_VEL
LIN {X 0,Y 587.348,Z 171.317,A -85,B 0,C 180,E1 -1454.258,E2 -1454.258} C_VEL
LIN {X 0,Y 587.341,Z 171.328,A -85,B 0,C 180,E1 -1457.407,E2 -1457.407} C_VEL
LIN {X 0,Y 587.319,Z 171.32,A -85,B 0,C 180,E1 -1460.306,E2 -1460.306} C_VEL
LIN {X 0,Y 587.313,Z 171.33,A -85,B 0,C 180,E1 -1463.259,E2 -1463.259} C_VEL
LIN {X 0,Y 587.321,Z 171.326,A -85,B 0,C 180,E1 -1465.518,E2 -1465.518} C_VEL
LIN {X 0,Y 587.34,Z 171.319,A -85,B 0,C 180,E1 -1467.818,E2 -1467.818} C_VEL
LIN {X 0,Y 587.322,Z 171.321,A -85,B 0,C 180,E1 -1470.509,E2 -1470.509} C_VEL
LIN {X 0,Y 587.331,Z 171.328,A -85,B 0,C 180,E1 -1473.112,E2 -1473.112} C_VEL
LIN {X 0,Y 587.29,Z 171.327,A -85,B 0,C 180,E1 -1475.538,E2 -1475.538} C_VEL
LIN {X 0,Y 587.328,Z 171.32,A -85,B 0,C 180,E1 -1477.839,E2 -1477.839} C_VEL
LIN {X 0,Y 587.305,Z 171.322,A -85,B 0,C 180,E1 -1480.255,E2 -1480.255} C_VEL
LIN {X 0,Y 587.301,Z 171.331,A -85,B 0,C 180,E1 -1483.118,E2 -1483.118} C_VEL
LIN {X 0,Y 587.308,Z 171.321,A -85,B 0,C 180,E1 -1486.049,E2 -1486.049} C_VEL
LIN {X 0,Y 587.332,Z 171.329,A -85,B 0,C 180,E1 -1488.926,E2 -1488.926} C_VEL
LIN {X 0,Y 587.316,Z 171.322,A -85,B 0,C 180,E1 -1491.521,E2 -1491.521} C_VEL
LIN {X 0,Y 587.284,Z 171.325,A -85,B 0,C 180,E1 -1494.1,E2 -1494.1} C_VEL
LIN {X 0,Y 587.333,Z 171.327,A -85,B 0,C 180,E1 -1496.89,E2 -1496.89} C_VEL
LIN {X 0,Y 587.317,Z 171.322,A -85,B 0,C 180,E1 -1499.494,E2 -1499.494} C_VEL
LIN {X 0,Y 587.339,Z 171.323,A -85,B 0,C 180,E1 -1502.31,E2 -1502.31} C_VEL
LIN {X 0,Y 587.303,Z 171.327,A -85,B 0,C 180,E1 -1505.24,E2 -1505.24} C_VEL
LIN {X 0,Y 587.354,Z 171.481,A -85,B 0,C 180,E1 -1505.995,E2 -1505.995} C_VEL
LIN {X 0,Y 588.117,Z 174.744,A -85,B 0,C 180,E1 -1506.402,E2 -1506.402} C_VEL
LIN {X 0,Y 588.008,Z 196.607,A -85,B 0,C 180,E1 -1508.793,E2 -1508.793} C_VEL
LIN {X 0,Y 587.791,Z 221.99,A -85,B 0,C 180,E1 -1511.528,E2 -1511.528} C_VEL
LIN {X 0,Y 587.63,Z 247.257,A -85,B 0,C 180,E1 -1514.212,E2 -1514.212} C_VEL
LIN {X 0,Y 587.494,Z 268.9,A -85,B 0,C 180,E1 -1516.467,E2 -1516.467} C_VEL
LIN {X 0,Y 587.846,Z 272.982,A -85,B 0,C 180,E1 -1516.541,E2 -1516.541} C_VEL
LIN {X 0,Y 587.725,Z 378.979,A -85,B 0,C 180,E1 -1517.856,E2 -1517.856} C_VEL
LIN {X 0,Y 587.682,Z 392.24,A -85,B 0,C 180,E1 -1518.161,E2 -1518.161} C_VEL
LIN {X 0,Y 587.627,Z 404.765,A -85,B 0,C 180,E1 -1518.591,E2 -1518.591} C_VEL
LIN {X 0,Y 587.54,Z 416.641,A -85,B 0,C 180,E1 -1519.141,E2 -1519.141} C_VEL
LIN {X 0,Y 587.469,Z 428.211,A -85,B 0,C 180,E1 -1519.837,E2 -1519.837} C_VEL
LIN {X 0,Y 587.393,Z 438.606,A -85,B 0,C 180,E1 -1520.618,E2 -1520.618} C_VEL
LIN {X 0,Y 587.321,Z 447.118,A -85,B 0,C 180,E1 -1521.398,E2 -1521.398} C_VEL
LIN {X 0,Y 587.273,Z 454.965,A -85,B 0,C 180,E1 -1522.263,E2 -1522.263} C_VEL
LIN {X 0,Y 587.23,Z 461.473,A -85,B 0,C 180,E1 -1523.127,E2 -1523.127} C_VEL
LIN {X 0,Y 587.236,Z 467.87,A -85,B 0,C 180,E1 -1524.162,E2 -1524.162} C_VEL
LIN {X 0,Y 587.147,Z 472.952,A -85,B 0,C 180,E1 -1525.194,E2 -1525.194} C_VEL
LIN {X 0,Y 587.213,Z 476.897,A -85,B 0,C 180,E1 -1526.226,E2 -1526.226} C_VEL
LIN {X 0,Y 587.132,Z 479.81,A -85,B 0,C 180,E1 -1527.256,E2 -1527.256} C_VEL
LIN {X 0,Y 587.141,Z 481.2,A -85,B 0,C 180,E1 -1527.943,E2 -1527.943} C_VEL
LIN {X 0,Y 587.14,Z 482.785,A -85,B 0,C 180,E1 -1529.315,E2 -1529.315} C_VEL
LIN {X 0,Y 587.137,Z 483,A -85,B 0,C 180,E1 -1530,E2 -1530} C_VEL
LIN {X 0,Y 587.147,Z 482.185,A -85,B 0,C 180,E1 -1531.372,E2 -1531.372} C_VEL
LIN {X 0,Y 587.141,Z 481.2,A -85,B 0,C 180,E1 -1532.058,E2 -1532.058} C_VEL
LIN {X 0,Y 587.132,Z 479.809,A -85,B 0,C 180,E1 -1532.745,E2 -1532.745} C_VEL
LIN {X 0,Y 587.213,Z 476.895,A -85,B 0,C 180,E1 -1533.775,E2 -1533.775} C_VEL
LIN {X 0,Y 587.147,Z 472.947,A -85,B 0,C 180,E1 -1534.807,E2 -1534.807} C_VEL
LIN {X 0,Y 587.217,Z 466.875,A -85,B 0,C 180,E1 -1536.012,E2 -1536.012} C_VEL
LIN {X 0,Y 587.245,Z 460.234,A -85,B 0,C 180,E1 -1537.047,E2 -1537.047} C_VEL
LIN {X 0,Y 587.3,Z 451.987,A -85,B 0,C 180,E1 -1538.083,E2 -1538.083} C_VEL
LIN {X 0,Y 587.344,Z 443.534,A -85,B 0,C 180,E1 -1538.949,E2 -1538.949} C_VEL
LIN {X 0,Y 587.421,Z 433.091,A -85,B 0,C 180,E1 -1539.817,E2 -1539.817} C_VEL
LIN {X 0,Y 587.493,Z 422.751,A -85,B 0,C 180,E1 -1540.512,E2 -1540.512} C_VEL
LIN {X 0,Y 587.585,Z 410.795,A -85,B 0,C 180,E1 -1541.149,E2 -1541.149} C_VEL
LIN {X 0,Y 587.64,Z 398.58,A -85,B 0,C 180,E1 -1541.64,E2 -1541.64} C_VEL
LIN {X 0,Y 587.729,Z 385.42,A -85,B 0,C 180,E1 -1542.014,E2 -1542.014} C_VEL
LIN {X 0,Y 587.767,Z 373.057,A -85,B 0,C 180,E1 -1542.232,E2 -1542.232} C_VEL
LIN {X 0,Y 587.808,Z 271.113,A -85,B 0,C 180,E1 -1543.483,E2 -1543.483} C_VEL
LIN {X 0,Y 587.491,Z 268.56,A -85,B 0,C 180,E1 -1543.556,E2 -1543.556} C_VEL
LIN {X 0,Y 587.667,Z 240.51,A -85,B 0,C 180,E1 -1546.501,E2 -1546.501} C_VEL
LIN {X 0,Y 587.858,Z 214.248,A -85,B 0,C 180,E1 -1549.302,E2 -1549.302} C_VEL
LIN {X 0,Y 588.063,Z 189.975,A -85,B 0,C 180,E1 -1551.93,E2 -1551.93} C_VEL
LIN {X 0,Y 588.12,Z 174.71,A -85,B 0,C 180,E1 -1553.599,E2 -1553.599} C_VEL
LIN {X 0,Y 587.347,Z 171.424,A -85,B 0,C 180,E1 -1554.006,E2 -1554.006} C_VEL
LIN {X 0,Y 587.309,Z 171.323,A -85,B 0,C 180,E1 -1556.28,E2 -1556.28} C_VEL
LIN {X 0,Y 587.344,Z 171.326,A -85,B 0,C 180,E1 -1559.132,E2 -1559.132} C_VEL
LIN {X 0,Y 587.317,Z 171.323,A -85,B 0,C 180,E1 -1561.831,E2 -1561.831} C_VEL
LIN {X 0,Y 587.334,Z 171.319,A -85,B 0,C 180,E1 -1564.345,E2 -1564.345} C_VEL
LIN {X 0,Y 587.342,Z 171.32,A -85,B 0,C 180,E1 -1567.608,E2 -1567.608} C_VEL
LIN {X 0,Y 587.307,Z 171.322,A -85,B 0,C 180,E1 -1570.255,E2 -1570.255} C_VEL
LIN {X 0,Y 587.304,Z 171.331,A -85,B 0,C 180,E1 -1573.117,E2 -1573.117} C_VEL
LIN {X 0,Y 587.3,Z 171.323,A -85,B 0,C 180,E1 -1576.047,E2 -1576.047} C_VEL
LIN {X 0,Y 587.334,Z 171.329,A -85,B 0,C 180,E1 -1578.925,E2 -1578.925} C_VEL
LIN {X 0,Y 587.32,Z 171.321,A -85,B 0,C 180,E1 -1581.52,E2 -1581.52} C_VEL
LIN {X 0,Y 587.289,Z 171.325,A -85,B 0,C 180,E1 -1584.099,E2 -1584.099} C_VEL
LIN {X 0,Y 587.338,Z 171.327,A -85,B 0,C 180,E1 -1586.889,E2 -1586.889} C_VEL
LIN {X 0,Y 587.321,Z 171.321,A -85,B 0,C 180,E1 -1589.493,E2 -1589.493} C_VEL
LIN {X 0,Y 587.343,Z 171.321,A -85,B 0,C 180,E1 -1592.309,E2 -1592.309} C_VEL
LIN {X 0,Y 587.35,Z 171.318,A -85,B 0,C 180,E1 -1595.241,E2 -1595.241} C_VEL
LIN {X 0,Y 587.317,Z 171.325,A -85,B 0,C 180,E1 -1598.225,E2 -1598.225} C_VEL
LIN {X 0,Y 587.347,Z 171.319,A -85,B 0,C 180,E1 -1601.151,E2 -1601.151} C_VEL
LIN {X 0,Y 587.316,Z 171.324,A -85,B 0,C 180,E1 -1604.024,E2 -1604.024} C_VEL
LIN {X 0,Y 587.348,Z 171.322,A -85,B 0,C 180,E1 -1606.154,E2 -1606.154} C_VEL
LIN {X 0,Y 587.34,Z 171.32,A -85,B 0,C 180,E1 -1608.962,E2 -1608.962} C_VEL
LIN {X 0,Y 587.339,Z 171.32,A -85,B 0,C 180,E1 -1611.744,E2 -1611.744} C_VEL
LIN {X 0,Y 587.356,Z 171.324,A -85,B 0,C 180,E1 -1614.507,E2 -1614.507} C_VEL
LIN {X 0,Y 587.367,Z 171.315,A -85,B 0,C 180,E1 -1617.256,E2 -1617.256} C_VEL
LIN {X 0,Y 587.378,Z 171.475,A -85,B 0,C 180,E1 -1619.978,E2 -1619.978} C_VEL
LIN {X 0,Y 587.442,Z 180.771,A -85,B 0,C 180,E1 -1621.714,E2 -1621.714} C_VEL
LIN {X 0,Y 587.388,Z 195.827,A -85,B 0,C 180,E1 -1624.46,E2 -1624.46} C_VEL
LIN {X 0,Y 587.292,Z 211.153,A -85,B 0,C 180,E1 -1627.218,E2 -1627.218} C_VEL
LIN {X 0,Y 587.272,Z 223.615,A -85,B 0,C 180,E1 -1629.406,E2 -1629.406} C_VEL
LIN {X 0,Y 587.474,Z 225.296,A -85,B 0,C 180,E1 -1629.467,E2 -1629.467} C_VEL
LIN {X 0,Y 587.541,Z 298.835,A -85,B 0,C 180,E1 -1630.378,E2 -1630.378} C_VEL
LIN {X 0,Y 587.178,Z 302.702,A -85,B 0,C 180,E1 -1630.436,E2 -1630.436} C_VEL
LIN {X 0,Y 585.831,Z 308.364,A -85,B 0,C 180,E1 -1630.545,E2 -1630.545} C_VEL
LIN {X 0,Y 583.865,Z 313.855,A -85,B 0,C 180,E1 -1630.67,E2 -1630.67} C_VEL
LIN {X 0,Y 581.087,Z 323.018,A -85,B 0,C 180,E1 -1630.973,E2 -1630.973} C_VEL
LIN {X 0,Y 580.429,Z 328.222,A -85,B 0,C 180,E1 -1631.21,E2 -1631.21} C_VEL
LIN {X 0,Y 580.315,Z 339.549,A -85,B 0,C 180,E1 -1631.881,E2 -1631.881} C_VEL
LIN {X 0,Y 580.234,Z 347.709,A -85,B 0,C 180,E1 -1632.504,E2 -1632.504} C_VEL
LIN {X 0,Y 580.213,Z 354.424,A -85,B 0,C 180,E1 -1633.127,E2 -1633.127} C_VEL
LIN {X 0,Y 580.163,Z 360.816,A -85,B 0,C 180,E1 -1633.842,E2 -1633.842} C_VEL
LIN {X 0,Y 580.13,Z 367.325,A -85,B 0,C 180,E1 -1634.738,E2 -1634.738} C_VEL
LIN {X 0,Y 580.081,Z 373.381,A -85,B 0,C 180,E1 -1635.819,E2 -1635.819} C_VEL
LIN {X 0,Y 580.056,Z 377.493,A -85,B 0,C 180,E1 -1636.83,E2 -1636.83} C_VEL
LIN {X 0,Y 580.046,Z 379.918,A -85,B 0,C 180,E1 -1637.632,E2 -1637.632} C_VEL
LIN {X 0,Y 580.034,Z 381.527,A -85,B 0,C 180,E1 -1638.362,E2 -1638.362} C_VEL
LIN {X 0,Y 580.056,Z 382.527,A -85,B 0,C 180,E1 -1639.095,E2 -1639.095} C_VEL
LIN {X 0,Y 580.016,Z 382.928,A -85,B 0,C 180,E1 -1639.832,E2 -1639.832} C_VEL
LIN {X 0,Y 580.041,Z 382.391,A -85,B 0,C 180,E1 -1641.099,E2 -1641.099} C_VEL
LIN {X 0,Y 580.036,Z 380.836,A -85,B 0,C 180,E1 -1642.062,E2 -1642.062} C_VEL
LIN {X 0,Y 580.069,Z 378.495,A -85,B 0,C 180,E1 -1642.957,E2 -1642.957} C_VEL
LIN {X 0,Y 580.076,Z 376.437,A -85,B 0,C 180,E1 -1643.566,E2 -1643.566} C_VEL
LIN {X 0,Y 580.093,Z 373.137,A -85,B 0,C 180,E1 -1644.325,E2 -1644.325} C_VEL
LIN {X 0,Y 580.122,Z 367.813,A -85,B 0,C 180,E1 -1645.28,E2 -1645.28} C_VEL
LIN {X 0,Y 580.141,Z 362.156,A -85,B 0,C 180,E1 -1646.083,E2 -1646.083} C_VEL
LIN {X 0,Y 580.192,Z 355.808,A -85,B 0,C 180,E1 -1646.821,E2 -1646.821} C_VEL
LIN {X 0,Y 580.235,Z 349.832,A -85,B 0,C 180,E1 -1647.404,E2 -1647.404} C_VEL
LIN {X 0,Y 580.305,Z 341.42,A -85,B 0,C 180,E1 -1648.077,E2 -1648.077} C_VEL
LIN {X 0,Y 580.363,Z 333.734,A -85,B 0,C 180,E1 -1648.576,E2 -1648.576} C_VEL
LIN {X 0,Y 580.417,Z 323.699,A -85,B 0,C 180,E1 -1649.094,E2 -1649.094} C_VEL
LIN {X 0,Y 580.534,Z 311.835,A -85,B 0,C 180,E1 -1649.537,E2 -1649.537} C_VEL
LIN {X 0,Y 580.519,Z 300.831,A -85,B 0,C 180,E1 -1649.797,E2 -1649.797} C_VEL
LIN {X 0,Y 580.568,Z 261.179,A -85,B 0,C 180,E1 -1650.307,E2 -1650.307} C_VEL
LIN {X 0,Y 580.436,Z 225.615,A -85,B 0,C 180,E1 -1650.748,E2 -1650.748} C_VEL
LIN {X 0,Y 580.252,Z 223.589,A -85,B 0,C 180,E1 -1650.818,E2 -1650.818} C_VEL
LIN {X 0,Y 580.3,Z 208.268,A -85,B 0,C 180,E1 -1653.553,E2 -1653.553} C_VEL
LIN {X 0,Y 580.423,Z 191.223,A -85,B 0,C 180,E1 -1656.669,E2 -1656.669} C_VEL
LIN {X 0,Y 580.506,Z 175.786,A -85,B 0,C 180,E1 -1659.53,E2 -1659.53} C_VEL
LIN {X 0,Y 580.33,Z 172.255,A -85,B 0,C 180,E1 -1660.216,E2 -1660.216} C_VEL
LIN {X 0,Y 580.275,Z 172.198,A -85,B 0,C 180,E1 -1662.706,E2 -1662.706} C_VEL
LIN {X 0,Y 580.269,Z 172.207,A -85,B 0,C 180,E1 -1665.609,E2 -1665.609} C_VEL
LIN {X 0,Y 580.297,Z 172.197,A -85,B 0,C 180,E1 -1668.233,E2 -1668.233} C_VEL
LIN {X 0,Y 580.274,Z 172.198,A -85,B 0,C 180,E1 -1670.965,E2 -1670.965} C_VEL
LIN {X 0,Y 580.28,Z 172.206,A -85,B 0,C 180,E1 -1673.597,E2 -1673.597} C_VEL
LIN {X 0,Y 580.314,Z 172.195,A -85,B 0,C 180,E1 -1676.145,E2 -1676.145} C_VEL
LIN {X 0,Y 580.275,Z 172.198,A -85,B 0,C 180,E1 -1678.614,E2 -1678.614} C_VEL
LIN {X 0,Y 580.292,Z 172.198,A -85,B 0,C 180,E1 -1681.024,E2 -1681.024} C_VEL
LIN {X 0,Y 580.327,Z 172.199,A -85,B 0,C 180,E1 -1683.658,E2 -1683.658} C_VEL
LIN {X 0,Y 580.278,Z 172.197,A -85,B 0,C 180,E1 -1686.442,E2 -1686.442} C_VEL
LIN {X 0,Y 580.274,Z 172.208,A -85,B 0,C 180,E1 -1689.437,E2 -1689.437} C_VEL
LIN {X 0,Y 580.267,Z 172.204,A -85,B 0,C 180,E1 -1691.645,E2 -1691.645} C_VEL
LIN {X 0,Y 580.277,Z 172.2,A -85,B 0,C 180,E1 -1693.825,E2 -1693.825} C_VEL
LIN {X 0,Y 580.324,Z 172.192,A -85,B 0,C 180,E1 -1695.983,E2 -1695.983} C_VEL
LIN {X 0,Y 580.303,Z 172.197,A -85,B 0,C 180,E1 -1698.826,E2 -1698.826} C_VEL
LIN {X 0,Y 580.332,Z 172.194,A -85,B 0,C 180,E1 -1701.644,E2 -1701.644} C_VEL
LIN {X 0,Y 580.326,Z 172.192,A -85,B 0,C 180,E1 -1704.44,E2 -1704.44} C_VEL
LIN {X 0,Y 580.344,Z 172.189,A -85,B 0,C 180,E1 -1707.918,E2 -1707.918} C_VEL
LIN {X 0,Y 580.357,Z 172.191,A -85,B 0,C 180,E1 -1710.693,E2 -1710.693} C_VEL
LIN {X 0,Y 580.284,Z 172.2,A -85,B 0,C 180,E1 -1713.471,E2 -1713.471} C_VEL
LIN {X 0,Y 580.328,Z 172.193,A -85,B 0,C 180,E1 -1715.559,E2 -1715.559} C_VEL
LIN {X 0,Y 580.326,Z 172.193,A -85,B 0,C 180,E1 -1718.356,E2 -1718.356} C_VEL
LIN {X 0,Y 580.296,Z 172.2,A -85,B 0,C 180,E1 -1721.191,E2 -1721.191} C_VEL
LIN {X 0,Y 580.323,Z 172.192,A -85,B 0,C 180,E1 -1724.016,E2 -1724.016} C_VEL
LIN {X 0,Y 580.308,Z 172.202,A -85,B 0,C 180,E1 -1726.913,E2 -1726.913} C_VEL
LIN {X 0,Y 580.301,Z 172.194,A -85,B 0,C 180,E1 -1729.822,E2 -1729.822} C_VEL
LIN {X 0,Y 580.292,Z 172.205,A -85,B 0,C 180,E1 -1732.802,E2 -1732.802} C_VEL
LIN {X 0,Y 580.304,Z 172.198,A -85,B 0,C 180,E1 -1735.079,E2 -1735.079} C_VEL
LIN {X 0,Y 580.315,Z 172.193,A -85,B 0,C 180,E1 -1737.863,E2 -1737.863} C_VEL
LIN {X 0,Y 580.287,Z 172.205,A -85,B 0,C 180,E1 -1740.696,E2 -1740.696} C_VEL
LIN {X 0,Y 580.299,Z 172.195,A -85,B 0,C 180,E1 -1743.316,E2 -1743.316} C_VEL
LIN {X 0,Y 580.32,Z 172.193,A -85,B 0,C 180,E1 -1745.767,E2 -1745.767} C_VEL
LIN {X 0,Y 580.282,Z 172.201,A -85,B 0,C 180,E1 -1748.146,E2 -1748.146} C_VEL
LIN {X 0,Y 580.294,Z 172.199,A -85,B 0,C 180,E1 -1750.843,E2 -1750.843} C_VEL
LIN {X 0,Y 580.28,Z 172.198,A -85,B 0,C 180,E1 -1753.656,E2 -1753.656} C_VEL
LIN {X 0,Y 580.269,Z 172.204,A -85,B 0,C 180,E1 -1756.609,E2 -1756.609} C_VEL
LIN {X 0,Y 580.296,Z 172.195,A -85,B 0,C 180,E1 -1759.157,E2 -1759.157} C_VEL
LIN {X 0,Y 580.283,Z 172.201,A -85,B 0,C 180,E1 -1761.926,E2 -1761.926} C_VEL
LIN {X 0,Y 580.299,Z 172.201,A -85,B 0,C 180,E1 -1764.456,E2 -1764.456} C_VEL
LIN {X 0,Y 580.284,Z 172.197,A -85,B 0,C 180,E1 -1766.975,E2 -1766.975} C_VEL
LIN {X 0,Y 580.301,Z 172.195,A -85,B 0,C 180,E1 -1769.426,E2 -1769.426} C_VEL
LIN {X 0,Y 580.312,Z 172.203,A -85,B 0,C 180,E1 -1772.137,E2 -1772.137} C_VEL
LIN {X 0,Y 580.313,Z 172.193,A -85,B 0,C 180,E1 -1775.269,E2 -1775.269} C_VEL
LIN {X 0,Y 580.266,Z 172.208,A -85,B 0,C 180,E1 -1777.948,E2 -1777.948} C_VEL
LIN {X 0,Y 580.31,Z 172.193,A -85,B 0,C 180,E1 -1780.914,E2 -1780.914} C_VEL
LIN {X 0,Y 580.273,Z 172.206,A -85,B 0,C 180,E1 -1783.826,E2 -1783.826} C_VEL
LIN {X 0,Y 580.317,Z 172.201,A -85,B 0,C 180,E1 -1785.983,E2 -1785.983} C_VEL
LIN {X 0,Y 580.323,Z 172.191,A -85,B 0,C 180,E1 -1788.828,E2 -1788.828} C_VEL
LIN {X 0,Y 580.325,Z 172.199,A -85,B 0,C 180,E1 -1791.644,E2 -1791.644} C_VEL
LIN {X 0,Y 580.312,Z 172.194,A -85,B 0,C 180,E1 -1794.44,E2 -1794.44} C_VEL
LIN {X 0,Y 580.336,Z 172.193,A -85,B 0,C 180,E1 -1797.224,E2 -1797.224} C_VEL
LIN {X 0,Y 580.34,Z 172.194,A -85,B 0,C 180,E1 -1800,E2 -1800} C_VEL
LIN {X 0,Y 580.33,Z 172.191,A -85,B 0,C 180,E1 -1802.777,E2 -1802.777} C_VEL
LIN {X 0,Y 580.318,Z 172.202,A -85,B 0,C 180,E1 -1805.56,E2 -1805.56} C_VEL
LIN {X 0,Y 580.301,Z 172.195,A -85,B 0,C 180,E1 -1808.357,E2 -1808.357} C_VEL
LIN {X 0,Y 580.292,Z 172.201,A -85,B 0,C 180,E1 -1811.192,E2 -1811.192} C_VEL
LIN {X 0,Y 580.31,Z 172.195,A -85,B 0,C 180,E1 -1814.018,E2 -1814.018} C_VEL
LIN {X 0,Y 580.305,Z 172.197,A -85,B 0,C 180,E1 -1816.914,E2 -1816.914} C_VEL
LIN {X 0,Y 580.279,Z 172.2,A -85,B 0,C 180,E1 -1819.824,E2 -1819.824} C_VEL
LIN {X 0,Y 580.264,Z 172.2,A -85,B 0,C 180,E1 -1822.053,E2 -1822.053} C_VEL
LIN {X 0,Y 580.297,Z 172.202,A -85,B 0,C 180,E1 -1825.081,E2 -1825.081} C_VEL
LIN {X 0,Y 580.292,Z 172.195,A -85,B 0,C 180,E1 -1828.186,E2 -1828.186} C_VEL
LIN {X 0,Y 580.275,Z 172.2,A -85,B 0,C 180,E1 -1830.695,E2 -1830.695} C_VEL
LIN {X 0,Y 580.277,Z 172.205,A -85,B 0,C 180,E1 -1833.314,E2 -1833.314} C_VEL
LIN {X 0,Y 580.239,Z 172.203,A -85,B 0,C 180,E1 -1835.757,E2 -1835.757} C_VEL
LIN {X 0,Y 580.279,Z 172.197,A -85,B 0,C 180,E1 -1838.147,E2 -1838.147} C_VEL
LIN {X 0,Y 580.291,Z 172.202,A -85,B 0,C 180,E1 -1840.844,E2 -1840.844} C_VEL
LIN {X 0,Y 580.264,Z 172.2,A -85,B 0,C 180,E1 -1843.66,E2 -1843.66} C_VEL
LIN {X 0,Y 580.264,Z 172.204,A -85,B 0,C 180,E1 -1846.611,E2 -1846.611} C_VEL
LIN {X 0,Y 580.287,Z 172.196,A -85,B 0,C 180,E1 -1849.731,E2 -1849.731} C_VEL
LIN {X 0,Y 580.284,Z 172.205,A -85,B 0,C 180,E1 -1852.732,E2 -1852.732} C_VEL
LIN {X 0,Y 580.288,Z 172.198,A -85,B 0,C 180,E1 -1855.444,E2 -1855.444} C_VEL
LIN {X 0,Y 580.296,Z 172.196,A -85,B 0,C 180,E1 -1857.971,E2 -1857.971} C_VEL
LIN {X 0,Y 580.281,Z 172.203,A -85,B 0,C 180,E1 -1861.024,E2 -1861.024} C_VEL
LIN {X 0,Y 580.266,Z 172.201,A -85,B 0,C 180,E1 -1863.672,E2 -1863.672} C_VEL
LIN {X 0,Y 580.313,Z 172.379,A -85,B 0,C 180,E1 -1865.828,E2 -1865.828} C_VEL
LIN {X 0,Y 581.347,Z 177.832,A -85,B 0,C 180,E1 -1866.489,E2 -1866.489} C_VEL
LIN {X 0,Y 581.067,Z 205.145,A -85,B 0,C 180,E1 -1869.467,E2 -1869.467} C_VEL
LIN {X 0,Y 580.784,Z 232.097,A -85,B 0,C 180,E1 -1872.392,E2 -1872.392} C_VEL
LIN {X 0,Y 580.594,Z 253.995,A -85,B 0,C 180,E1 -1874.736,E2 -1874.736} C_VEL
LIN {X 0,Y 580.515,Z 268.901,A -85,B 0,C 180,E1 -1876.301,E2 -1876.301} C_VEL
LIN {X 0,Y 580.936,Z 274.771,A -85,B 0,C 180,E1 -1876.4,E2 -1876.4} C_VEL
LIN {X 0,Y 580.808,Z 378.979,A -85,B 0,C 180,E1 -1877.709,E2 -1877.709} C_VEL
LIN {X 0,Y 580.737,Z 392.24,A -85,B 0,C 180,E1 -1878.018,E2 -1878.018} C_VEL
LIN {X 0,Y 580.677,Z 405.51,A -85,B 0,C 180,E1 -1878.481,E2 -1878.481} C_VEL
LIN {X 0,Y 580.563,Z 416.639,A -85,B 0,C 180,E1 -1879.009,E2 -1879.009} C_VEL
LIN {X 0,Y 580.447,Z 428.211,A -85,B 0,C 180,E1 -1879.713,E2 -1879.713} C_VEL
LIN {X 0,Y 580.345,Z 438.607,A -85,B 0,C 180,E1 -1880.503,E2 -1880.503} C_VEL
LIN {X 0,Y 580.271,Z 447.118,A -85,B 0,C 180,E1 -1881.293,E2 -1881.293} C_VEL
LIN {X 0,Y 580.221,Z 454.965,A -85,B 0,C 180,E1 -1882.169,E2 -1882.169} C_VEL
LIN {X 0,Y 580.153,Z 462.654,A -85,B 0,C 180,E1 -1883.222,E2 -1883.222} C_VEL
LIN {X 0,Y 580.139,Z 469.683,A -85,B 0,C 180,E1 -1884.439,E2 -1884.439} C_VEL
LIN {X 0,Y 580.108,Z 474.374,A -85,B 0,C 180,E1 -1885.484,E2 -1885.484} C_VEL
LIN {X 0,Y 580.123,Z 477.959,A -85,B 0,C 180,E1 -1886.528,E2 -1886.528} C_VEL
LIN {X 0,Y 580.043,Z 479.809,A -85,B 0,C 180,E1 -1887.223,E2 -1887.223} C_VEL
LIN {X 0,Y 580.04,Z 481.199,A -85,B 0,C 180,E1 -1887.917,E2 -1887.917} C_VEL
LIN {X 0,Y 580.04,Z 482.785,A -85,B 0,C 180,E1 -1889.306,E2 -1889.306} C_VEL
LIN {X 0,Y 580.037,Z 483,A -85,B 0,C 180,E1 -1890,E2 -1890} C_VEL
LIN {X 0,Y 580.046,Z 482.186,A -85,B 0,C 180,E1 -1891.389,E2 -1891.389} C_VEL
LIN {X 0,Y 580.04,Z 481.199,A -85,B 0,C 180,E1 -1892.084,E2 -1892.084} C_VEL
LIN {X 0,Y 580.043,Z 479.809,A -85,B 0,C 180,E1 -1892.778,E2 -1892.778} C_VEL
LIN {X 0,Y 580.11,Z 476.894,A -85,B 0,C 180,E1 -1893.821,E2 -1893.821} C_VEL
LIN {X 0,Y 580.053,Z 472.947,A -85,B 0,C 180,E1 -1894.866,E2 -1894.866} C_VEL
LIN {X 0,Y 580.139,Z 466.874,A -85,B 0,C 180,E1 -1896.085,E2 -1896.085} C_VEL
LIN {X 0,Y 580.185,Z 460.235,A -85,B 0,C 180,E1 -1897.133,E2 -1897.133} C_VEL
LIN {X 0,Y 580.251,Z 451.987,A -85,B 0,C 180,E1 -1898.182,E2 -1898.182} C_VEL
LIN {X 0,Y 580.308,Z 443.534,A -85,B 0,C 180,E1 -1899.059,E2 -1899.059} C_VEL
LIN {X 0,Y 580.425,Z 433.093,A -85,B 0,C 180,E1 -1899.936,E2 -1899.936} C_VEL
LIN {X 0,Y 580.497,Z 422.749,A -85,B 0,C 180,E1 -1900.64,E2 -1900.64} C_VEL
LIN {X 0,Y 580.598,Z 411.226,A -85,B 0,C 180,E1 -1901.265,E2 -1901.265} C_VEL
LIN {X 0,Y 580.68,Z 398.461,A -85,B 0,C 180,E1 -1901.785,E2 -1901.785} C_VEL
LIN {X 0,Y 580.779,Z 385.418,A -85,B 0,C 180,E1 -1902.16,E2 -1902.16} C_VEL
LIN {X 0,Y 580.836,Z 373.057,A -85,B 0,C 180,E1 -1902.38,E2 -1902.38} C_VEL
LIN {X 0,Y 580.794,Z 271.113,A -85,B 0,C 180,E1 -1903.649,E2 -1903.649} C_VEL
LIN {X 0,Y 580.517,Z 268.561,A -85,B 0,C 180,E1 -1903.722,E2 -1903.722} C_VEL
LIN {X 0,Y 580.73,Z 240.51,A -85,B 0,C 180,E1 -1906.704,E2 -1906.704} C_VEL
LIN {X 0,Y 581.019,Z 211.873,A -85,B 0,C 180,E1 -1909.797,E2 -1909.797} C_VEL
LIN {X 0,Y 581.237,Z 186.305,A -85,B 0,C 180,E1 -1912.576,E2 -1912.576} C_VEL
LIN {X 0,Y 581.295,Z 177.539,A -85,B 0,C 180,E1 -1913.515,E2 -1913.515} C_VEL
LIN {X 0,Y 580.308,Z 172.336,A -85,B 0,C 180,E1 -1914.126,E2 -1914.126} C_VEL
LIN {X 0,Y 580.257,Z 172.203,A -85,B 0,C 180,E1 -1916.625,E2 -1916.625} C_VEL
LIN {X 0,Y 580.278,Z 172.208,A -85,B 0,C 180,E1 -1919.305,E2 -1919.305} C_VEL
LIN {X 0,Y 580.286,Z 172.197,A -85,B 0,C 180,E1 -1922.201,E2 -1922.201} C_VEL
LIN {X 0,Y 580.284,Z 172.2,A -85,B 0,C 180,E1 -1924.697,E2 -1924.697} C_VEL
LIN {X 0,Y 580.289,Z 172.204,A -85,B 0,C 180,E1 -1927.269,E2 -1927.269} C_VEL
LIN {X 0,Y 580.287,Z 172.197,A -85,B 0,C 180,E1 -1930.269,E2 -1930.269} C_VEL
LIN {X 0,Y 580.268,Z 172.203,A -85,B 0,C 180,E1 -1933.389,E2 -1933.389} C_VEL
LIN {X 0,Y 580.243,Z 172.203,A -85,B 0,C 180,E1 -1936.338,E2 -1936.338} C_VEL
LIN {X 0,Y 580.296,Z 172.201,A -85,B 0,C 180,E1 -1939.156,E2 -1939.156} C_VEL
LIN {X 0,Y 580.287,Z 172.196,A -85,B 0,C 180,E1 -1941.928,E2 -1941.928} C_VEL
LIN {X 0,Y 580.25,Z 172.205,A -85,B 0,C 180,E1 -1944.452,E2 -1944.452} C_VEL
LIN {X 0,Y 580.289,Z 172.203,A -85,B 0,C 180,E1 -1946.975,E2 -1946.975} C_VEL
LIN {X 0,Y 580.283,Z 172.198,A -85,B 0,C 180,E1 -1949.424,E2 -1949.424} C_VEL
LIN {X 0,Y 580.292,Z 172.198,A -85,B 0,C 180,E1 -1952.143,E2 -1952.143} C_VEL
LIN {X 0,Y 580.321,Z 172.194,A -85,B 0,C 180,E1 -1955.27,E2 -1955.27} C_VEL
LIN {X 0,Y 580.269,Z 172.2,A -85,B 0,C 180,E1 -1957.947,E2 -1957.947} C_VEL
LIN {X 0,Y 580.298,Z 172.2,A -85,B 0,C 180,E1 -1960.913,E2 -1960.913} C_VEL
LIN {X 0,Y 580.27,Z 172.2,A -85,B 0,C 180,E1 -1963.825,E2 -1963.825} C_VEL
LIN {X 0,Y 580.317,Z 172.196,A -85,B 0,C 180,E1 -1965.983,E2 -1965.983} C_VEL
LIN {X 0,Y 580.306,Z 172.198,A -85,B 0,C 180,E1 -1968.827,E2 -1968.827} C_VEL
LIN {X 0,Y 580.308,Z 172.195,A -85,B 0,C 180,E1 -1971.643,E2 -1971.643} C_VEL
LIN {X 0,Y 580.321,Z 172.201,A -85,B 0,C 180,E1 -1974.44,E2 -1974.44} C_VEL
LIN {X 0,Y 580.334,Z 172.192,A -85,B 0,C 180,E1 -1977.223,E2 -1977.223} C_VEL
LIN {X 0,Y 580.346,Z 172.334,A -85,B 0,C 180,E1 -1979.913,E2 -1979.913} C_VEL
LIN {X 0,Y 580.485,Z 180.241,A -85,B 0,C 180,E1 -1981.387,E2 -1981.387} C_VEL
LIN {X 0,Y 580.385,Z 193.386,A -85,B 0,C 180,E1 -1983.818,E2 -1983.818} C_VEL
LIN {X 0,Y 580.297,Z 209.347,A -85,B 0,C 180,E1 -1986.733,E2 -1986.733} C_VEL
LIN {X 0,Y 580.234,Z 223.676,A -85,B 0,C 180,E1 -1989.279,E2 -1989.279} C_VEL
LIN {X 0,Y 580.611,Z 226.857,A -85,B 0,C 180,E1 -1989.361,E2 -1989.361} C_VEL
LIN {X 0,Y 580.533,Z 300.372,A -85,B 0,C 180,E1 -1990.286,E2 -1990.286} C_VEL
LIN {X 0,Y 580.486,Z 310.098,A -85,B 0,C 180,E1 -1990.507,E2 -1990.507} C_VEL
LIN {X 0,Y 580.467,Z 321.572,A -85,B 0,C 180,E1 -1990.899,E2 -1990.899} C_VEL
LIN {X 0,Y 580.429,Z 328.222,A -85,B 0,C 180,E1 -1991.21,E2 -1991.21} C_VEL
LIN {X 0,Y 579.714,Z 333.469,A -85,B 0,C 180,E1 -1991.472,E2 -1991.472} C_VEL
LIN {X 0,Y 576.793,Z 341.623,A -85,B 0,C 180,E1 -1991.954,E2 -1991.954} C_VEL
LIN {X 0,Y 573.875,Z 349.142,A -85,B 0,C 180,E1 -1992.529,E2 -1992.529} C_VEL
LIN {X 0,Y 573.167,Z 353.388,A -85,B 0,C 180,E1 -1992.934,E2 -1992.934} C_VEL
LIN {X 0,Y 573.121,Z 359.918,A -85,B 0,C 180,E1 -1993.654,E2 -1993.654} C_VEL
LIN {X 0,Y 573.065,Z 365.112,A -85,B 0,C 180,E1 -1994.34,E2 -1994.34} C_VEL
LIN {X 0,Y 573.076,Z 368.915,A -85,B 0,C 180,E1 -1994.924,E2 -1994.924} C_VEL
LIN {X 0,Y 572.993,Z 372.864,A -85,B 0,C 180,E1 -1995.654,E2 -1995.654} C_VEL
LIN {X 0,Y 572.981,Z 376.048,A -85,B 0,C 180,E1 -1996.386,E2 -1996.386} C_VEL
LIN {X 0,Y 572.979,Z 378.569,A -85,B 0,C 180,E1 -1997.12,E2 -1997.12} C_VEL
LIN {X 0,Y 572.946,Z 380.506,A -85,B 0,C 180,E1 -1997.858,E2 -1997.858} C_VEL
LIN {X 0,Y 572.965,Z 382.624,A -85,B 0,C 180,E1 -1999.182,E2 -1999.182} C_VEL
LIN {X 0,Y 572.944,Z 382.996,A -85,B 0,C 180,E1 -2000.087,E2 -2000.087} C_VEL
LIN {X 0,Y 572.962,Z 382.253,A -85,B 0,C 180,E1 -2001.216,E2 -2001.216} C_VEL
LIN {X 0,Y 572.947,Z 380.236,A -85,B 0,C 180,E1 -2002.349,E2 -2002.349} C_VEL
LIN {X 0,Y 572.987,Z 378.115,A -85,B 0,C 180,E1 -2003.11,E2 -2003.11} C_VEL
LIN {X 0,Y 573.006,Z 375.313,A -85,B 0,C 180,E1 -2003.875,E2 -2003.875} C_VEL
LIN {X 0,Y 573.035,Z 370.759,A -85,B 0,C 180,E1 -2004.828,E2 -2004.828} C_VEL
LIN {X 0,Y 573.065,Z 366.022,A -85,B 0,C 180,E1 -2005.613,E2 -2005.613} C_VEL
LIN {X 0,Y 573.093,Z 360.753,A -85,B 0,C 180,E1 -2006.332,E2 -2006.332} C_VEL
LIN {X 0,Y 573.122,Z 355.071,A -85,B 0,C 180,E1 -2006.982,E2 -2006.982} C_VEL
LIN {X 0,Y 573.204,Z 347.819,A -85,B 0,C 180,E1 -2007.67,E2 -2007.67} C_VEL
LIN {X 0,Y 573.25,Z 340.228,A -85,B 0,C 180,E1 -2008.261,E2 -2008.261} C_VEL
LIN {X 0,Y 573.381,Z 330.752,A -85,B 0,C 180,E1 -2008.857,E2 -2008.857} C_VEL
LIN {X 0,Y 573.452,Z 320.278,A -85,B 0,C 180,E1 -2009.355,E2 -2009.355} C_VEL
LIN {X 0,Y 573.523,Z 309.907,A -85,B 0,C 180,E1 -2009.706,E2 -2009.706} C_VEL
LIN {X 0,Y 573.53,Z 300.15,A -85,B 0,C 180,E1 -2009.928,E2 -2009.928} C_VEL
LIN {X 0,Y 573.593,Z 227.18,A -85,B 0,C 180,E1 -2010.858,E2 -2010.858} C_VEL
LIN {X 0,Y 573.212,Z 223.985,A -85,B 0,C 180,E1 -2010.924,E2 -2010.924} C_VEL
LIN {X 0,Y 573.153,Z 223.236,A -85,B 0,C 180,E1 -2010.997,E2 -2010.997} C_VEL
LIN {X 0,Y 573.235,Z 207.273,A -85,B 0,C 180,E1 -2013.906,E2 -2013.906} C_VEL
LIN {X 0,Y 573.416,Z 192.227,A -85,B 0,C 180,E1 -2016.69,E2 -2016.69} C_VEL
LIN {X 0,Y 573.49,Z 176.52,A -85,B 0,C 180,E1 -2019.587,E2 -2019.587} C_VEL
LIN {X 0,Y 573.305,Z 173.109,A -85,B 0,C 180,E1 -2020.26,E2 -2020.26} C_VEL
LIN {X 0,Y 573.234,Z 173.079,A -85,B 0,C 180,E1 -2023.359,E2 -2023.359} C_VEL
LIN {X 0,Y 573.242,Z 173.076,A -85,B 0,C 180,E1 -2026.331,E2 -2026.331} C_VEL
LIN {X 0,Y 573.237,Z 173.075,A -85,B 0,C 180,E1 -2028.543,E2 -2028.543} C_VEL
LIN {X 0,Y 573.239,Z 173.078,A -85,B 0,C 180,E1 -2031.298,E2 -2031.298} C_VEL
LIN {X 0,Y 573.243,Z 173.078,A -85,B 0,C 180,E1 -2034.014,E2 -2034.014} C_VEL
LIN {X 0,Y 573.268,Z 173.071,A -85,B 0,C 180,E1 -2036.518,E2 -2036.518} C_VEL
LIN {X 0,Y 573.226,Z 173.079,A -85,B 0,C 180,E1 -2039.118,E2 -2039.118} C_VEL
LIN {X 0,Y 573.236,Z 173.083,A -85,B 0,C 180,E1 -2041.435,E2 -2041.435} C_VEL
LIN {X 0,Y 573.288,Z 173.073,A -85,B 0,C 180,E1 -2043.811,E2 -2043.811} C_VEL
LIN {X 0,Y 573.231,Z 173.076,A -85,B 0,C 180,E1 -2046.134,E2 -2046.134} C_VEL
LIN {X 0,Y 573.25,Z 173.079,A -85,B 0,C 180,E1 -2049.173,E2 -2049.173} C_VEL
LIN {X 0,Y 573.223,Z 173.086,A -85,B 0,C 180,E1 -2051.411,E2 -2051.411} C_VEL
LIN {X 0,Y 573.25,Z 173.078,A -85,B 0,C 180,E1 -2053.621,E2 -2053.621} C_VEL
LIN {X 0,Y 573.272,Z 173.073,A -85,B 0,C 180,E1 -2055.807,E2 -2055.807} C_VEL
LIN {X 0,Y 573.261,Z 173.074,A -85,B 0,C 180,E1 -2058.745,E2 -2058.745} C_VEL
LIN {X 0,Y 573.288,Z 173.073,A -85,B 0,C 180,E1 -2061.54,E2 -2061.54} C_VEL
LIN {X 0,Y 573.295,Z 173.068,A -85,B 0,C 180,E1 -2064.371,E2 -2064.371} C_VEL
LIN {X 0,Y 573.314,Z 173.065,A -85,B 0,C 180,E1 -2067.892,E2 -2067.892} C_VEL
LIN {X 0,Y 573.328,Z 173.067,A -85,B 0,C 180,E1 -2070.702,E2 -2070.702} C_VEL
LIN {X 0,Y 573.301,Z 173.073,A -85,B 0,C 180,E1 -2072.81,E2 -2072.81} C_VEL
LIN {X 0,Y 573.295,Z 173.068,A -85,B 0,C 180,E1 -2075.628,E2 -2075.628} C_VEL
LIN {X 0,Y 573.282,Z 173.071,A -85,B 0,C 180,E1 -2078.459,E2 -2078.459} C_VEL
LIN {X 0,Y 573.268,Z 173.074,A -85,B 0,C 180,E1 -2081.311,E2 -2081.311} C_VEL
LIN {X 0,Y 573.278,Z 173.073,A -85,B 0,C 180,E1 -2084.424,E2 -2084.424} C_VEL
LIN {X 0,Y 573.254,Z 173.077,A -85,B 0,C 180,E1 -2087.111,E2 -2087.111} C_VEL
LIN {X 0,Y 573.248,Z 173.074,A -85,B 0,C 180,E1 -2090.076,E2 -2090.076} C_VEL
LIN {X 0,Y 573.229,Z 173.079,A -85,B 0,C 180,E1 -2093.099,E2 -2093.099} C_VEL
LIN {X 0,Y 573.253,Z 173.073,A -85,B 0,C 180,E1 -2095.409,E2 -2095.409} C_VEL
LIN {X 0,Y 573.259,Z 173.073,A -85,B 0,C 180,E1 -2098.031,E2 -2098.031} C_VEL
LIN {X 0,Y 573.233,Z 173.08,A -85,B 0,C 180,E1 -2100.883,E2 -2100.883} C_VEL
LIN {X 0,Y 573.282,Z 173.069,A -85,B 0,C 180,E1 -2103.528,E2 -2103.528} C_VEL
LIN {X 0,Y 573.255,Z 173.075,A -85,B 0,C 180,E1 -2106.048,E2 -2106.048} C_VEL
LIN {X 0,Y 573.241,Z 173.08,A -85,B 0,C 180,E1 -2108.701,E2 -2108.701} C_VEL
LIN {X 0,Y 573.246,Z 173.073,A -85,B 0,C 180,E1 -2111.595,E2 -2111.595} C_VEL
LIN {X 0,Y 573.231,Z 173.084,A -85,B 0,C 180,E1 -2114.333,E2 -2114.333} C_VEL
LIN {X 0,Y 573.232,Z 173.075,A -85,B 0,C 180,E1 -2117.358,E2 -2117.358} C_VEL
LIN {X 0,Y 573.242,Z 173.082,A -85,B 0,C 180,E1 -2120.393,E2 -2120.393} C_VEL
LIN {X 0,Y 573.248,Z 173.073,A -85,B 0,C 180,E1 -2123.078,E2 -2123.078} C_VEL
LIN {X 0,Y 573.266,Z 173.073,A -85,B 0,C 180,E1 -2125.672,E2 -2125.672} C_VEL
LIN {X 0,Y 573.243,Z 173.084,A -85,B 0,C 180,E1 -2128.185,E2 -2128.185} C_VEL
LIN {X 0,Y 573.263,Z 173.074,A -85,B 0,C 180,E1 -2130.634,E2 -2130.634} C_VEL
LIN {X 0,Y 573.242,Z 173.074,A -85,B 0,C 180,E1 -2133.024,E2 -2133.024} C_VEL
LIN {X 0,Y 573.267,Z 173.072,A -85,B 0,C 180,E1 -2135.366,E2 -2135.366} C_VEL
LIN {X 0,Y 573.223,Z 173.08,A -85,B 0,C 180,E1 -2138.419,E2 -2138.419} C_VEL
LIN {X 0,Y 573.271,Z 173.071,A -85,B 0,C 180,E1 -2140.728,E2 -2140.728} C_VEL
LIN {X 0,Y 573.25,Z 173.078,A -85,B 0,C 180,E1 -2143.622,E2 -2143.622} C_VEL
LIN {X 0,Y 573.264,Z 173.08,A -85,B 0,C 180,E1 -2145.807,E2 -2145.807} C_VEL
LIN {X 0,Y 573.275,Z 173.07,A -85,B 0,C 180,E1 -2148.734,E2 -2148.734} C_VEL
LIN {X 0,Y 573.281,Z 173.074,A -85,B 0,C 180,E1 -2151.541,E2 -2151.541} C_VEL
LIN {X 0,Y 573.279,Z 173.071,A -85,B 0,C 180,E1 -2154.372,E2 -2154.372} C_VEL
LIN {X 0,Y 573.297,Z 173.074,A -85,B 0,C 180,E1 -2157.893,E2 -2157.893} C_VEL
LIN {X 0,Y 573.322,Z 173.064,A -85,B 0,C 180,E1 -2160.703,E2 -2160.703} C_VEL
LIN {X 0,Y 573.234,Z 173.083,A -85,B 0,C 180,E1 -2163.515,E2 -2163.515} C_VEL
LIN {X 0,Y 573.283,Z 173.078,A -85,B 0,C 180,E1 -2165.629,E2 -2165.629} C_VEL
LIN {X 0,Y 573.267,Z 173.077,A -85,B 0,C 180,E1 -2167.751,E2 -2167.751} C_VEL
LIN {X 0,Y 573.257,Z 173.072,A -85,B 0,C 180,E1 -2170.597,E2 -2170.597} C_VEL
LIN {X 0,Y 573.255,Z 173.073,A -85,B 0,C 180,E1 -2172.749,E2 -2172.749} C_VEL
LIN {X 0,Y 573.226,Z 173.078,A -85,B 0,C 180,E1 -2174.92,E2 -2174.92} C_VEL
LIN {X 0,Y 573.234,Z 173.078,A -85,B 0,C 180,E1 -2177.849,E2 -2177.849} C_VEL
LIN {X 0,Y 573.234,Z 173.076,A -85,B 0,C 180,E1 -2180.078,E2 -2180.078} C_VEL
LIN {X 0,Y 573.229,Z 173.075,A -85,B 0,C 180,E1 -2182.338,E2 -2182.338} C_VEL
LIN {X 0,Y 573.24,Z 173.082,A -85,B 0,C 180,E1 -2185.411,E2 -2185.411} C_VEL
LIN {X 0,Y 573.244,Z 173.074,A -85,B 0,C 180,E1 -2188.03,E2 -2188.03} C_VEL
LIN {X 0,Y 573.223,Z 173.081,A -85,B 0,C 180,E1 -2190.883,E2 -2190.883} C_VEL
LIN {X 0,Y 573.235,Z 173.079,A -85,B 0,C 180,E1 -2193.521,E2 -2193.521} C_VEL
LIN {X 0,Y 573.208,Z 173.078,A -85,B 0,C 180,E1 -2196.052,E2 -2196.052} C_VEL
LIN {X 0,Y 573.233,Z 173.079,A -85,B 0,C 180,E1 -2198.703,E2 -2198.703} C_VEL
LIN {X 0,Y 573.222,Z 173.078,A -85,B 0,C 180,E1 -2201.593,E2 -2201.593} C_VEL
LIN {X 0,Y 573.224,Z 173.077,A -85,B 0,C 180,E1 -2204.335,E2 -2204.335} C_VEL
LIN {X 0,Y 573.221,Z 173.08,A -85,B 0,C 180,E1 -2207.361,E2 -2207.361} C_VEL
LIN {X 0,Y 573.239,Z 173.077,A -85,B 0,C 180,E1 -2210.393,E2 -2210.393} C_VEL
LIN {X 0,Y 573.229,Z 173.082,A -85,B 0,C 180,E1 -2213.077,E2 -2213.077} C_VEL
LIN {X 0,Y 573.257,Z 173.073,A -85,B 0,C 180,E1 -2215.672,E2 -2215.672} C_VEL
LIN {X 0,Y 573.233,Z 173.077,A -85,B 0,C 180,E1 -2218.185,E2 -2218.185} C_VEL
LIN {X 0,Y 573.238,Z 173.084,A -85,B 0,C 180,E1 -2220.634,E2 -2220.634} C_VEL
LIN {X 0,Y 573.208,Z 173.086,A -85,B 0,C 180,E1 -2223.023,E2 -2223.023} C_VEL
LIN {X 0,Y 573.277,Z 173.277,A -85,B 0,C 180,E1 -2225.656,E2 -2225.656} C_VEL
LIN {X 0,Y 574.43,Z 178.741,A -85,B 0,C 180,E1 -2226.328,E2 -2226.328} C_VEL
LIN {X 0,Y 574.173,Z 204.949,A -85,B 0,C 180,E1 -2229.209,E2 -2229.209} C_VEL
LIN {X 0,Y 573.882,Z 230.412,A -85,B 0,C 180,E1 -2231.988,E2 -2231.988} C_VEL
LIN {X 0,Y 573.646,Z 253.995,A -85,B 0,C 180,E1 -2234.546,E2 -2234.546} C_VEL
LIN {X 0,Y 573.521,Z 268.902,A -85,B 0,C 180,E1 -2236.131,E2 -2236.131} C_VEL
LIN {X 0,Y 574.036,Z 274.771,A -85,B 0,C 180,E1 -2236.234,E2 -2236.234} C_VEL
LIN {X 0,Y 573.885,Z 378.979,A -85,B 0,C 180,E1 -2237.558,E2 -2237.558} C_VEL
LIN {X 0,Y 573.793,Z 392.24,A -85,B 0,C 180,E1 -2237.87,E2 -2237.87} C_VEL
LIN {X 0,Y 573.688,Z 405.169,A -85,B 0,C 180,E1 -2238.325,E2 -2238.325} C_VEL
LIN {X 0,Y 573.59,Z 416.724,A -85,B 0,C 180,E1 -2238.879,E2 -2238.879} C_VEL
LIN {X 0,Y 573.439,Z 428.208,A -85,B 0,C 180,E1 -2239.586,E2 -2239.586} C_VEL
LIN {X 0,Y 573.332,Z 438.609,A -85,B 0,C 180,E1 -2240.386,E2 -2240.386} C_VEL
LIN {X 0,Y 573.24,Z 447.118,A -85,B 0,C 180,E1 -2241.185,E2 -2241.185} C_VEL
LIN {X 0,Y 573.16,Z 454.965,A -85,B 0,C 180,E1 -2242.072,E2 -2242.072} C_VEL
LIN {X 0,Y 573.072,Z 462.958,A -85,B 0,C 180,E1 -2243.186,E2 -2243.186} C_VEL
LIN {X 0,Y 573.07,Z 469.683,A -85,B 0,C 180,E1 -2244.37,E2 -2244.37} C_VEL
LIN {X 0,Y 573.028,Z 474.374,A -85,B 0,C 180,E1 -2245.428,E2 -2245.428} C_VEL
LIN {X 0,Y 573.022,Z 477.959,A -85,B 0,C 180,E1 -2246.485,E2 -2246.485} C_VEL
LIN {X 0,Y 572.959,Z 479.809,A -85,B 0,C 180,E1 -2247.188,E2 -2247.188} C_VEL
LIN {X 0,Y 572.946,Z 482.186,A -85,B 0,C 180,E1 -2248.595,E2 -2248.595} C_VEL
LIN {X 0,Y 572.938,Z 483,A -85,B 0,C 180,E1 -2250,E2 -2250} C_VEL
LIN {X 0,Y 572.946,Z 482.185,A -85,B 0,C 180,E1 -2251.406,E2 -2251.406} C_VEL
LIN {X 0,Y 572.94,Z 481.198,A -85,B 0,C 180,E1 -2252.109,E2 -2252.109} C_VEL
LIN {X 0,Y 572.959,Z 479.809,A -85,B 0,C 180,E1 -2252.813,E2 -2252.813} C_VEL
LIN {X 0,Y 573.015,Z 476.894,A -85,B 0,C 180,E1 -2253.868,E2 -2253.868} C_VEL
LIN {X 0,Y 572.963,Z 472.947,A -85,B 0,C 180,E1 -2254.926,E2 -2254.926} C_VEL
LIN {X 0,Y 573.065,Z 466.874,A -85,B 0,C 180,E1 -2256.161,E2 -2256.161} C_VEL
LIN {X 0,Y 573.12,Z 460.234,A -85,B 0,C 180,E1 -2257.221,E2 -2257.221} C_VEL
LIN {X 0,Y 573.201,Z 451.987,A -85,B 0,C 180,E1 -2258.284,E2 -2258.284} C_VEL
LIN {X 0,Y 573.287,Z 443.534,A -85,B 0,C 180,E1 -2259.171,E2 -2259.171} C_VEL
LIN {X 0,Y 573.431,Z 433.092,A -85,B 0,C 180,E1 -2260.059,E2 -2260.059} C_VEL
LIN {X 0,Y 573.515,Z 422.764,A -85,B 0,C 180,E1 -2260.77,E2 -2260.77} C_VEL
LIN {X 0,Y 573.629,Z 411.578,A -85,B 0,C 180,E1 -2261.386,E2 -2261.386} C_VEL
LIN {X 0,Y 573.716,Z 399.757,A -85,B 0,C 180,E1 -2261.885,E2 -2261.885} C_VEL
LIN {X 0,Y 573.857,Z 386.332,A -85,B 0,C 180,E1 -2262.286,E2 -2262.286} C_VEL
LIN {X 0,Y 573.902,Z 373.057,A -85,B 0,C 180,E1 -2262.532,E2 -2262.532} C_VEL
LIN {X 0,Y 574.049,Z 272.902,A -85,B 0,C 180,E1 -2263.79,E2 -2263.79} C_VEL
